# B&R Automation Studio project EFI (part 8)

### Stacker.typ
```iecst
TYPE
	StackerCtrlStatus_enum :
		(
		STACKERCTRL_STOPPED,
		STACKERCTRL_STOPPING,
		STACKERCTRL_PREPARING,
		STACKERCTRL_PREPARED,
		STACKERCTRL_PAUSING,
		STACKERCTRL_PAUSED,
		STACKERCTRL_STARTING,
		STACKERCTRL_WORKING,
		STACKERCTRL_CONTROLSTOPPING
		);
	StackerStatus_enum :
		(
		STACKER_TURNED_OFF,
		STACKER_INIT,
		STACKER_PREPARING,
		STACKER_READY,
		STACKER_WORKING,
		STACKER_FAULTED
		);
	StackerType_enum :
		(
		STACKERTY_UNDEFINED,
		STACKERTY_FULL_S,
		STACKERTY_BUNDLE_S
		);
	StackerInputs_typ : 	STRUCT
		xError : BOOL;
		xRunning : BOOL;
		xReadyToStack : BOOL;
		xFeedInterrupt : BOOL;
		xStackSuccess : BOOL;
		xRejectSuccess : BOOL;
		xModelInput : ARRAY[0..2]OF BOOL;
		Comms : StackerCommsInputs_typ;
		xStackerPresent : BOOL;
		xNoPowered : BOOL;
	END_STRUCT;
	StackerOutputs_typ : 	STRUCT
		xRun : BOOL;
		xStackEject : BOOL;
		xEjectRejectStack : BOOL;
		xPrepareToStack : BOOL;
		xRejectSheet : BOOL;
		xCleanBelts : BOOL; (*Command to empty stacker's belts*)
	END_STRUCT;
	StackerAlarms_typ : 	STRUCT
		xError : BOOL;
		xFeedInterrupt : BOOL;
		xAlrOutAutomatic : BOOL;
		xAnyAlarm : BOOL;
		xNotRemote : BOOL;
		xCriticalAlarm : BOOL;
		xWarningAlarm : BOOL;
		xNoStackerPresent : BOOL;
		xCommsError : BOOL;
		xNoPowered : BOOL;
		xBeltsStopped : BOOL;
		xRejectNoAvailable : BOOL;
		xStopRequest : BOOL; (*Stop request from Dryer when physical stop button is pressed*)
	END_STRUCT;
	StackerParametersSw_typ : 	STRUCT
		xEnabled : BOOL;
		iStackHeight : UINT;
		iStackBoardsNum : UINT;
		xStackMode : BOOL; (*(0 - Stack per number of boards, 1 - Stack per height)*)
	END_STRUCT;
	StackerParametersHw_typ : 	STRUCT
		xRejectEjectionAvailable : BOOL; (*stacker has the possibility to eject rejected boards automatically*)
		xThereIsReject : BOOL; (*Stacker has reject device*)
		rMaxSpeed : REAL := 100.0; (*Maximum speed allowed in m/min*)
		iMaxMediaWidth : UINT; (*Maximum media width allowed in mm*)
		iMinMediaWidth : UINT; (*Minimum media width allowed in mm*)
		iMinMediaThickness : UINT; (*Maximum media length allowed in mm*)
		iMaxMediaThickness : UINT; (*Minimum media length allowed in mm*)
		iMaxMediaLength : UINT; (*Maximum media length allowed in mm*)
		iMinMediaLength : UINT; (*Minimum media length allowed in mm*)
		iRejectAdjustmentDistance : INT; (*Distance in cm from beginning of the Stacker to Reject Position. Positive inside Stacker. Negative previous to Stacker*)
		iDistanceToReject : INT; (*Distance measured from "iRejectAdjusmentDistance" to reject belt start of the stacker. Physically from sensor at stacker's entry to the reject belt*)
		iMinStackHeight : UINT;
		iMaxStackHeight : UINT;
		iMinStackBoards : UINT;
		iMaxStackBoards : UINT;
		rStackerLength : REAL;
		xDoubleLineAllowed : BOOL; (*Active when allows double line printing*)
	END_STRUCT;
	StackerParameters_typ : 	STRUCT
		xInstalled : BOOL;
		xSimulationMode : BOOL; (*Defined by the configuration in Automation Studio*)
		xCommsOK : BOOL;
		xAlrPresent : BOOL;
		LineState : LineStatus_enum;
		xLineInAuto : BOOL;
		xInRemote : BOOL;
		Media : StackerMediaParameters;
		rSpeedSetPoint : REAL;
		rMediaLength : REAL;
		xPreviousDeviceStopped : BOOL;
		xDoubleLine : BOOL;
		LineStatusSummary : LineControlStatusSummarized;
		Hw : StackerParametersHw_typ;
		xActiveSlaveDiagnosis : BOOL;
	END_STRUCT;
	StackerCommands_typ : 	STRUCT
		xStart : BOOL; (*Edge commands. Reseted when managed*)
		xPrepare : BOOL; (*Edge commands. Reseted when managed*)
		xPause : BOOL; (*Edge commands. Reseted when managed*)
		xControlStop : BOOL; (*Edge commands. Reseted when managed*)
		xStop : BOOL; (*Edge commands. Reseted when managed*)
		xStartTransport : BOOL; (*Edge commands. Reseted when managed*)
		xResetAlarms : BOOL; (*Edge commands. Reseted when managed*)
		xRejectSheet : BOOL;
		xEjectPileStack : BOOL; (*Edge commands. Reseted when managed*)
		xCleanBelts : BOOL; (*Edge commands. Reseted when managed*)
		xEjectRejectStack : BOOL; (*Edge commands. Reseted when managed*)
	END_STRUCT;
	StackerOrders_typ : 	STRUCT
		xHoldReject : BOOL; (*While the signal is 1, the reject remains activated.*)
		xRejectSheet : BOOL;
		xDisableWriteBlock : BOOL; (*No read/write of channels of block (Modbus)*)
		xDisableReadBlock : BOOL;
	END_STRUCT;
	StackerDeviceStatus_typ : 	STRUCT
		xTurnedOff : BOOL;
		xInit : BOOL;
		xPreparing : BOOL;
		xReadyToStack : BOOL;
		xStacking : BOOL;
		xStackEjecting : BOOL;
		xFaulted : BOOL;
		xNotRemote : BOOL;
	END_STRUCT;
	StackerStatus_typ : 	STRUCT
		iModel : UINT; (*Model of the Device*)
		Version : EFI_version_typ;
		CtrlStatus : StackerCtrlStatus_enum;
		DeviceStatus : StackerStatus_enum;
		Device : StackerDeviceStatus_typ;
		xBeltEmpty : BOOL;
		StackerType : StackerType_enum;
		Comms : StackerCommsStatus_typ;
	END_STRUCT;
	Stacker_typ : 	STRUCT
		Inputs : StackerInputs_typ;
		Outputs : StackerOutputs_typ;
		Alarms : StackerAlarms_typ;
		ParSw : StackerParametersSw_typ;
		Parameters : StackerParameters_typ;
		Commands : StackerCommands_typ; (*Just Edge commands*)
		Orders : StackerOrders_typ;
		Status : StackerStatus_typ;
		Comms : StackerCommsOutputs_typ;
	END_STRUCT;
	StackerCommsInputs_typ : 	STRUCT
		xCommsOK : BOOL; (*Modbus communications are working properly*)
		xRemote : BOOL; (*(0: local; 1: remote)*)
		xErrorActive : BOOL; (*Any critical alarm activated*)
		xWarningActive : BOOL; (*Any warning alarm activated*)
		xOnline : BOOL; (*Modbus communications OK in stacker's side*)
		xNewFormat : BOOL; (*New box format. Please, empty stack*)
		xSerie : BOOL; (*Machine serie, SerA = 1 / SerB =0*)
		xBeltsEmpty : BOOL; (*Belts with no boards*)
		xRejectAvailable : BOOL; (*(1 = Reject Available; 0 = Reject not available)*)
		xEmergencyStopNotAcknowledged : BOOL; (*Safety alarm not acknowledge on stacker's HMI*)
		xInWorkingPosition : BOOL; (*Stacker positioned*)
		xStackExit : BOOL; (*Pile leaving*)
		xStopDemand : BOOL; (*Boards sending request*)
		xStackerEmpty : BOOL; (*Stacker and belt with no boards*)
		xStackReady : BOOL; (*Pile ready to be extracted*)
		iVersion1 : INT; (*Machine platform (Nozomi = 1)*)
		iVersion2 : INT; (*Machine project (C18000 = 0 / C14000 = 1)*)
		iVersion3 : INT; (*Hardware version*)
		iVersion4 : INT; (*Sotfware version*)
		iStatus : INT; (*Status word*)
		iAlarmWord1 : INT; (*Status word*)
		iAlarmWord2 : INT; (*Status word*)
		iAlarmWord3 : INT; (*Status word*)
		iAlarmWord4 : INT; (*Status word*)
		iAlarmWord5 : INT; (*Status word*)
		iAlarmWord6 : INT; (*Status word*)
		iAlarmWord7 : INT; (*Status word*)
		iAlarmWord8 : INT; (*Status word*)
		iAlarmWord9 : INT; (*Status word*)
		iAlarmWord10 : INT; (*Status word*)
		uiTransportSpeed : UINT;
		uiNumBoardsInCurrentPile : INT;
		uiCurrentPileHeigh : INT;
	END_STRUCT;
	StackerCommsOutputs_typ : 	STRUCT
		iControl : INT; (*Status word*)
		xBelEmpty : BOOL; (*Edge commands. Reseted when managed*)
		xResetAlarms : BOOL;
		xNewBoardParameters : BOOL; (*Pulse to let know board paramters have changed*)
		xCleanBelts : BOOL; (*Command to empty stacker's belts*)
		xEndCycle : BOOL; (*Controlled stop with pile stacked output*)
		xLastBox : BOOL; (*Signal for indicate the last box of the current pile*)
	END_STRUCT;
	StackerMediaParameters : 	STRUCT
		rThickness : REAL; (*Tile thickness to print from gui in mm*)
		rWidth : REAL; (*Board's width in mm*)
		rGap : REAL; (*Gap between boards in mm*)
		rLength : REAL; (*Board's length in mm*)
		rOffsetRegisterL1 : REAL; (*Board's width in mm*)
		rOffsetRegisterL2 : REAL; (*Board's width in mm*)
	END_STRUCT;
	StackerCommsStatus_typ : 	STRUCT
		xModuleOk : BOOL;
		ModSlaveState : UINT;
		LastError : UINT;
		LastErrorBlockNum : UINT;
		xStopButtonPressed : BOOL;
		ActOverloadError : BOOL;
		ActModbusError : BOOL;
		ActSlvConError : BOOL;
		ActRefreshError : BOOL;
		ActInternalError : BOOL;
		ActConfError : BOOL;
		HistOverloadError : BOOL;
		HistModbusError : BOOL;
		HistSlvConError : BOOL;
		HistRefreshError : BOOL;
		HistInternalError : BOOL;
		HistConfError : BOOL;
		ModbusErrorCnt : UINT;
		ModbusConErrorCnt : UINT;
		ModbusPktRefreshTimeoutCnt : UINT;
		ModbusPktPendPerSec : UINT;
		ModbusMeanResponseTime : UINT;
	END_STRUCT;
END_TYPE
```

### Program Logical/ExtPack/_Ancillaries/StackerCtrl/StackerSim/StackerSim_v1/StackerSim (IEC)

#### StackerSim.st - Init, cyclic, exit code
```iecst
PROGRAM _INIT

	Stacker ACCESS ADR(gStacker);
	SimStacker ACCESS ADR(gSimStacker);

	Stacker.Status.Comms.xModuleOk := TRUE;
	Stacker.Inputs.Comms.xBeltsEmpty:=TRUE;

END_PROGRAM

PROGRAM _CYCLIC
	(* Insert code here *)
	Stacker ACCESS ADR(gStacker);
	SimStacker ACCESS ADR(gSimStacker);

	Stacker.Inputs.xStackerPresent:=TRUE;
	Stacker.Inputs.Comms.xRemote := TRUE;

	Stacker.Inputs.xError:=SimStacker.Commands.CreateError;

	tonReady.IN:= Stacker.Outputs.xPrepareToStack;
	tonReady.PT:= T#2s;
	tonReady();
	Stacker.Inputs.xReadyToStack:=tonReady.Q;

	tonRun.IN:= Stacker.Inputs.xReadyToStack AND Stacker.Outputs.xRun;
	tonRun.PT:= T#1s;
	tonRun();
	Stacker.Inputs.xRunning:=tonRun.Q AND NOT SimStacker.Commands.StopBelts;

END_PROGRAM
```

### Library Logical/ExtPack/_Comms/ModbusComms/ModbusComms_v1/Libraries/BRSE_MB (ANSIC)

#### BRSE_MB.var
```iecst
VAR CONSTANT
	BRSE_MB_MAX_COILS : UINT := 2000;
	BRSE_MB_MAX_DISCRETE_INPUTS : UINT := 2000;
	BRSE_MB_MAX_HOLDING_REG_READ : USINT := 125;
	BRSE_MB_MAX_INPUT_REG_READ : USINT := 125;
	BRSE_MB_MAX_HOLDING_REG_WRITE : USINT := 100;
	BRSE_MB_MAX_COILS_WRITE : UINT := 800;
	BRSE_MB_ERR_REFERENCE : UINT := 20002;
	BRSE_MB_ERR_UNIT_ALLOCATED : UINT := 20001;
	BRSE_MB_ERR_ILLEGAL_FUNCTION : UINT := 1;
	BRSE_MB_ERR_ILLEGAL_DATA_ADDRESS : USINT := 2;
	BRSE_MB_ERR_ILLEGAL_DATA_VALUE : USINT := 3;
	BRSE_MB_ERR_ILLEGAL_RESPONSE_LEN : UINT := 4;
	BRSE_MB_READ_COILS : UINT := 16#01;
	BRSE_MB_READ_DISCRETE_INPUTS : UINT := 16#02;
	BRSE_MB_READ_HOLDING_REGISTERS : UINT := 16#03;
	BRSE_MB_READ_HOLDING_REG_4BYTE : UINT := 16#30;
	BRSE_MB_READ_INPUT_REGISTERS : UINT := 16#04;
	BRSE_MB_WRITE_SINGLE_COIL : UINT := 16#05;
	BRSE_MB_WRITE_SINGLE_REGISTER : UINT := 16#06;
	BRSE_MB_WRITE_MULTIPLE_COILS : UINT := 16#0F;
	BRSE_MB_WRITE_MULTIPLE_REGISTERS : UINT := 16#10;
	BRSE_MB_WRITE_MULTIPLE_REG_4BYTE : UINT := 16#31;
	BRSE_MB_ON : UINT := 16#FF00;
	BRSE_MB_OFF : UINT := 16#0000;
	BRSE_MB_MAX_UNIT_ID : USINT := 255;
	BRSE_MB_INTEL : USINT := 0; (* The server/client uses the Intel format *)
	BRSE_MB_MOTOROLA : USINT := 1; (* The server/client uses the Motorola format *)
	MB_QUEUE_SIZE : UINT := 50; (*Design parameter. Number of commands that can be queued for each client. If >= number of FB (using ClientID), race conditions (starvation?) is prevented*)
	MB_MAX_CLIENTS : USINT := 10; (*Design parameter. Maximum ClientID that can be used.*)
	MB_ERR_CLIENT_ALLOCATED : UINT := 20003; (*Error code: Queue for this client id has already been allocated*)
	MB_ERR_CLIENT_NOT_ALLOCATED : UINT := 20004; (*A request was requested from a client which hasn't been allocated*)
	MB_ERR_BUFFER : UINT := 20005; (*Buffer is too small for request or buffer address is 0*)
	MB_ERR_QUEUE_FULL : UINT := 20006;
	MB_ERR_INTERNAL : UINT := 20007;
	MB_ERR_PROTOCOL : UINT := 20008;
	MB_ERR_QUANTITY : UINT := 20009; (*Input quantity error (too big or 0)*)
	MB_ERR_CLIENT : UINT := 20010; (*Request dropped out of queue. Warm restart with remanent FUB? (Client queue is volatile)*)
	MB_ERR_CONNECTION : UINT := 20011; (*Request could not be executed: connection error or no response from server*)
END_VAR
```

#### BRSE_MB.fun
```iecst
FUNCTION MB_GetClient : UDINT (*Debug function. Returns pointer to MB_Client_typ*)
	VAR_INPUT
		ClientID : USINT;
	END_VAR
END_FUNCTION

FUNCTION BRSE_MB_Alloc : UDINT (*Allocate memory for internal data (configuration etc.). Returns error code or pointer.*)
	VAR_INPUT
		Unit : USINT; (*Unit (card id) to allocate. 0-254*)
		MaxCoils : UINT; (*Max 2000*)
		MaxHoldingRegisters : UINT; (*Max 2000*)
		MaxDiscreteInputs : UINT; (*Max 125*)
		MaxInputRegisters : UINT; (*Max 125*)
	END_VAR
END_FUNCTION

FUNCTION BRSE_MB_Coil : UINT
	VAR_INPUT
		Unit : USINT;
		Reference : UINT; (*Variable index (0-2000)*)
		VariableAddress : UDINT;
	END_VAR
END_FUNCTION

FUNCTION BRSE_MB_HoldingRegister : UINT
	VAR_INPUT
		Unit : USINT;
		Reference : UINT; (*Variable index (0-2000)*)
		VariableAddress : UDINT;
	END_VAR
END_FUNCTION

FUNCTION BRSE_MB_4ByteHoldingRegister : UINT
	VAR_INPUT
		Unit : USINT;
		Reference : UINT; (*Variable index (0-2000)*)
		VariableAddress : UDINT;
	END_VAR
END_FUNCTION

FUNCTION BRSE_MB_InputRegister : UINT
	VAR_INPUT
		Unit : USINT;
		Reference : UINT; (*Variable index (0-2000)*)
		VariableAddress : UDINT;
	END_VAR
END_FUNCTION

FUNCTION BRSE_MB_DiscreteInput : UINT
	VAR_INPUT
		Unit : USINT;
		Reference : UINT; (*Variable index (0-2000)*)
		VariableAddress : UDINT;
	END_VAR
END_FUNCTION

FUNCTION_BLOCK BRSE_MB_Server
	VAR_INPUT
		Unit : USINT;
		ClientFormat : USINT;
		InputBuffer : ARRAY[0..254] OF USINT;
	END_VAR
	VAR_OUTPUT
		OutputBuffer : ARRAY[0..254] OF USINT;
		Status : UINT;
		BufferLength : USINT; (*Total number of bytes in output buffer*)
	END_VAR
	VAR
		Request : BRSE_MB_Request_typ;
	END_VAR
END_FUNCTION_BLOCK

FUNCTION MB_AllocClient : UDINT
	VAR_INPUT
		ClientID : USINT;
	END_VAR
END_FUNCTION

FUNCTION_BLOCK MB_PollCoils
	VAR_INPUT
		ClientID : USINT;
		Enable : BOOL;
		Quantity : UINT;
		PollInterval : UDINT; (*Interval in ms between the read requests*)
		VariablesAddress : UDINT;
		StartAddress : UINT;
		Unit : USINT; (*Unit in the server*)
	END_VAR
	VAR_OUTPUT
		UpdateDone : BOOL;
		Busy : BOOL;
		Active : BOOL;
		Error : BOOL;
		ErrorID : UINT;
		Status : UINT;
	END_VAR
	VAR
		Step : UINT;
		RequestStatus : UINT;
		InternalStatus : UINT;
		RTInfo_0 : RTInfo;
		CycleTimeMs : UDINT; (*Task cycle time in ms*)
		ElapsedTime : UDINT; (*Ms since last request*)
	END_VAR
END_FUNCTION_BLOCK

FUNCTION_BLOCK MB_PollDiscreteInputs
	VAR_INPUT
		ClientID : USINT;
		Enable : BOOL;
		Quantity : UINT;
		PollInterval : UDINT; (*Interval in ms between the read requests*)
		VariablesAddress : UDINT;
		StartAddress : UINT;
		Unit : USINT; (*Unit in the server*)
	END_VAR
	VAR_OUTPUT
		UpdateDone : BOOL;
		Busy : BOOL;
		Active : BOOL;
		Error : BOOL;
		ErrorID : UINT;
		Status : UINT;
	END_VAR
	VAR
		Step : UINT;
		RequestStatus : UINT;
		InternalStatus : UINT;
		RTInfo_0 : RTInfo;
		CycleTimeMs : UDINT; (*Task cycle time in ms*)
		ElapsedTime : UDINT; (*Ms since last request*)
	END_VAR
END_FUNCTION_BLOCK

FUNCTION_BLOCK MB_PollHoldingRegisters
	VAR_INPUT
		ClientID : USINT;
		Enable : BOOL;
		Quantity : UINT;
		PollInterval : UDINT; (*Interval in ms between the read requests*)
		VariablesAddress : UDINT;
		StartAddress : UINT;
		Unit : USINT; (*Unit in the server*)
	END_VAR
	VAR_OUTPUT
		UpdateDone : BOOL;
		Busy : BOOL;
		Active : BOOL;
		Error : BOOL;
		ErrorID : UINT;
		Status : UINT;
	END_VAR
	VAR
		Step : UINT;
		RequestStatus : UINT;
		InternalStatus : UINT;
		RTInfo_0 : RTInfo;
		CycleTimeMs : UDINT; (*Task cycle time in ms*)
		ElapsedTime : UDINT; (*Ms since last request*)
	END_VAR
END_FUNCTION_BLOCK

FUNCTION_BLOCK MB_Poll4ByteHoldingRegisters
	VAR_INPUT
		ClientID : USINT;
		Enable : BOOL;
		Quantity : UINT;
		PollInterval : UDINT; (*Interval in ms between the read requests*)
		VariablesAddress : UDINT;
		StartAddress : UINT;
		Unit : USINT; (*Unit in the server*)
	END_VAR
	VAR_OUTPUT
		UpdateDone : BOOL;
		Busy : BOOL;
		Active : BOOL;
		Error : BOOL;
		ErrorID : UINT;
		Status : UINT;
	END_VAR
	VAR
		Step : UINT;
		RequestStatus : UINT;
		InternalStatus : UINT;
		RTInfo_0 : RTInfo;
		CycleTimeMs : UDINT; (*Task cycle time in ms*)
		ElapsedTime : UDINT; (*Ms since last request*)
	END_VAR
END_FUNCTION_BLOCK

FUNCTION_BLOCK MB_PollInputRegisters
	VAR_INPUT
		ClientID : USINT;
		Enable : BOOL;
		Quantity : UINT;
		PollInterval : UDINT; (*Interval in ms between the read requests*)
		VariablesAddress : UDINT;
		StartAddress : UINT;
		Unit : USINT; (*Unit in the server*)
	END_VAR
	VAR_OUTPUT
		UpdateDone : BOOL;
		Busy : BOOL;
		Active : BOOL;
		Error : BOOL;
		ErrorID : UINT;
		Status : UINT;
	END_VAR
	VAR
		Step : UINT;
		RequestStatus : UINT;
		InternalStatus : UINT;
		RTInfo_0 : RTInfo;
		CycleTimeMs : UDINT; (*Task cycle time in ms*)
		ElapsedTime : UDINT; (*Ms since last request*)
	END_VAR
END_FUNCTION_BLOCK

FUNCTION_BLOCK MB_PushCoils
	VAR_INPUT
		ClientID : USINT;
		Enable : BOOL;
		Quantity : UINT;
		PushInterval : UDINT; (*Interval in ms between the write requests*)
		VariablesAddress : UDINT;
		StartAddress : UINT;
		Unit : USINT; (*Unit in the server*)
	END_VAR
	VAR_OUTPUT
		UpdateDone : BOOL;
		Busy : BOOL;
		Active : BOOL;
		Error : BOOL;
		ErrorID : UINT;
		Status : UINT;
	END_VAR
	VAR
		Step : UINT;
		RequestStatus : UINT;
		InternalStatus : UINT;
		RTInfo_0 : RTInfo;
		CycleTimeMs : UDINT; (*Task cycle time in ms*)
		ElapsedTime : UDINT; (*Ms since last request*)
	END_VAR
END_FUNCTION_BLOCK

FUNCTION_BLOCK MB_PushHoldingRegisters
	VAR_INPUT
		ClientID : USINT;
		Enable : BOOL;
		Quantity : UINT;
		PushInterval : UDINT; (*Interval in ms between the write requests*)
		VariablesAddress : UDINT;
		StartAddress : UINT;
		Unit : USINT; (*Unit in the server*)
	END_VAR
	VAR_OUTPUT
		UpdateDone : BOOL;
		Busy : BOOL;
		Active : BOOL;
		Error : BOOL;
		ErrorID : UINT;
		Status : UINT;
	END_VAR
	VAR
		Step : UINT;
		RequestStatus : UINT;
		InternalStatus : UINT;
		RTInfo_0 : RTInfo;
		CycleTimeMs : UDINT; (*Task cycle time in ms*)
		ElapsedTime : UDINT; (*Ms since last request*)
	END_VAR
END_FUNCTION_BLOCK

FUNCTION_BLOCK MB_Push4ByteHoldingRegisters
	VAR_INPUT
		ClientID : USINT;
		Enable : BOOL;
		Quantity : UINT;
		PushInterval : UDINT; (*Interval in ms between the write requests*)
		VariablesAddress : UDINT;
		StartAddress : UINT;
		Unit : USINT; (*Unit in the server*)
	END_VAR
	VAR_OUTPUT
		UpdateDone : BOOL;
		Busy : BOOL;
		Active : BOOL;
		Error : BOOL;
		ErrorID : UINT;
		Status : UINT;
	END_VAR
	VAR
		Step : UINT;
		RequestStatus : UINT;
		InternalStatus : UINT;
		RTInfo_0 : RTInfo;
		CycleTimeMs : UDINT; (*Task cycle time in ms*)
		ElapsedTime : UDINT; (*Ms since last request*)
	END_VAR
END_FUNCTION_BLOCK

FUNCTION_BLOCK MB_ReadCoils
	VAR_INPUT
		ClientID : USINT;
		Execute : BOOL;
		Quantity : UINT;
		VariablesAddress : UDINT;
		StartAddress : UINT;
		Unit : USINT; (*Unit in the server*)
	END_VAR
	VAR_OUTPUT
		Busy : BOOL;
		Done : BOOL;
		Error : BOOL;
		ErrorID : UINT;
		Status : UINT;
	END_VAR
	VAR
		Step : UINT;
		RequestStatus : UINT;
		InternalStatus : UINT;
	END_VAR
END_FUNCTION_BLOCK

FUNCTION_BLOCK MB_ReadDiscreteInputs
	VAR_INPUT
		ClientID : USINT;
		Execute : BOOL;
		Quantity : UINT;
		VariablesAddress : UDINT;
		StartAddress : UINT;
		Unit : USINT; (*Unit in the server*)
	END_VAR
	VAR_OUTPUT
		Busy : BOOL;
		Done : BOOL;
		Error : BOOL;
		ErrorID : UINT;
		Status : UINT;
	END_VAR
	VAR
		Step : UINT;
		RequestStatus : UINT;
		InternalStatus : UINT;
	END_VAR
END_FUNCTION_BLOCK

FUNCTION_BLOCK MB_ReadHoldingRegisters
	VAR_INPUT
		ClientID : USINT;
		Execute : BOOL;
		Quantity : UINT;
		VariablesAddress : UDINT;
		StartAddress : UINT;
		Unit : USINT; (*Unit in the server*)
	END_VAR
	VAR_OUTPUT
		Busy : BOOL;
		Done : BOOL;
		Error : BOOL;
		ErrorID : UINT;
		Status : UINT;
	END_VAR
	VAR
		Step : UINT;
		RequestStatus : UINT;
		InternalStatus : UINT;
	END_VAR
END_FUNCTION_BLOCK

FUNCTION_BLOCK MB_Read4ByteHoldingRegisters
	VAR_INPUT
		ClientID : USINT;
		Execute : BOOL;
		Quantity : UINT;
		VariablesAddress : UDINT;
		StartAddress : UINT;
		Unit : USINT; (*Unit in the server*)
	END_VAR
	VAR_OUTPUT
		Busy : BOOL;
		Done : BOOL;
		Error : BOOL;
		ErrorID : UINT;
		Status : UINT;
	END_VAR
	VAR
		Step : UINT;
		RequestStatus : UINT;
		InternalStatus : UINT;
	END_VAR
END_FUNCTION_BLOCK

FUNCTION_BLOCK MB_ReadInputRegisters
	VAR_INPUT
		ClientID : USINT;
		Execute : BOOL;
		Quantity : UINT;
		VariablesAddress : UDINT;
		StartAddress : UINT;
		Unit : USINT; (*Unit in the server*)
	END_VAR
	VAR_OUTPUT
		Busy : BOOL;
		Done : BOOL;
		Error : BOOL;
		ErrorID : UINT;
		Status : UINT;
	END_VAR
	VAR
		Step : UINT;
		RequestStatus : UINT;
		InternalStatus : UINT;
	END_VAR
END_FUNCTION_BLOCK

FUNCTION_BLOCK MB_WriteCoils
	VAR_INPUT
		ClientID : USINT;
		Execute : BOOL;
		Quantity : UINT;
		VariablesAddress : UDINT;
		StartAddress : UINT;
		Unit : USINT; (*Unit in the server*)
	END_VAR
	VAR_OUTPUT
		Busy : BOOL;
		Done : BOOL;
		Error : BOOL;
		ErrorID : UINT;
		Status : UINT;
	END_VAR
	VAR
		Step : UINT;
		RequestStatus : UINT;
		InternalStatus : UINT;
	END_VAR
END_FUNCTION_BLOCK

FUNCTION_BLOCK MB_WriteHoldingRegisters
	VAR_INPUT
		ClientID : USINT;
		Execute : BOOL;
		Quantity : UINT;
		VariablesAddress : UDINT;
		StartAddress : UINT;
		Unit : USINT; (*Unit in the server*)
	END_VAR
	VAR_OUTPUT
		Busy : BOOL;
		Done : BOOL;
		Error : BOOL;
		ErrorID : UINT;
		Status : UINT;
	END_VAR
	VAR
		Step : UINT;
		RequestStatus : UINT;
		InternalStatus : UINT;
	END_VAR
END_FUNCTION_BLOCK

FUNCTION_BLOCK MB_Write4ByteHoldingRegisters
	VAR_INPUT
		ClientID : USINT;
		Execute : BOOL;
		Quantity : UINT;
		VariablesAddress : UDINT;
		StartAddress : UINT;
		Unit : USINT; (*Unit in the server*)
	END_VAR
	VAR_OUTPUT
		Busy : BOOL;
		Done : BOOL;
		Error : BOOL;
		ErrorID : UINT;
		Status : UINT;
	END_VAR
	VAR
		Step : UINT;
		RequestStatus : UINT;
		InternalStatus : UINT;
	END_VAR
END_FUNCTION_BLOCK

FUNCTION_BLOCK MB_CreateClientRequest (*This function block is used only internally and from the BRSE_MBT library (os other libraries processing the request queue)*)
	VAR_INPUT
		ClientID : USINT;
		ServerFormat : USINT;
		AdrByteBuffer : UDINT; (*Address to byte buffer where to create the request*)
		ByteBufferLen : UINT; (*Length of the byte buffer*)
	END_VAR
	VAR_OUTPUT
		RequestBufferLen : UINT; (*Length of the created modbus request. 0 means that no requests are in queue.*)
		Status : UINT; (*Error code. 0 if successful.*)
		Unit : USINT; (*Unit in the server*)
	END_VAR
END_FUNCTION_BLOCK

FUNCTION_BLOCK MB_PutClientResponse (*This function block is used only internally and from the BRSE_MBT library (os other libraries processing the request queue)*)
	VAR_INPUT
		ClientID : USINT;
		ServerFormat : USINT;
		AdrByteBuffer : UDINT;
		ByteBufferLen : UINT;
	END_VAR
	VAR_OUTPUT
		Status : UINT;
	END_VAR
	VAR
		ResponseInfo : BRSE_MB_Request_typ;
		Step : UINT;
	END_VAR
END_FUNCTION_BLOCK

FUNCTION MB_AckClientRequest : UINT (*This function is used only internally and from the BRSE_MBT library (os other libraries processing the request queue)*)
	VAR_INPUT
		ClientID : USINT;
		ReturnStatus : UINT;
	END_VAR
END_FUNCTION
```

#### Example.c
```c
/*!
\page Example

\section Example
For an example on how to use this library. Please take a look in the help for BRSE_MBT or BRSE_MBR.

*/
```

#### MB_Client.c
```c
/*! \file MB_Client.c */

#include <bur/plctypes.h>
#include "BRSE_MB.h"
#include "BRSE_MB_Main.h"

/***************************/
/* Necessary byte swapping */
/***************************/
#ifdef _SG4
	#define SWAPUINT	swapUINT
	#define SWAPINT		swapINT
#else
	#define SWAPUINT
	#define SWAPINT
#endif

#define	BUSY				65535

MB_ClientStruct_typ gMB_ClientInternal;

UDINT MB_GetClient(USINT ClientID)
{
	return gMB_ClientInternal.pClients[ClientID];
}

/*! \interface MB_AllocClient
	\brief Client: Allocate memory for internal data (request queue etc.)
	\param ClientID Client ID to allocate.
	\retval DataAddress DataAddress to internal structure. Used for debug purposes. Same value as MB_GetClient returns.
*/
UDINT MB_AllocClient(unsigned char ClientID)
{
	UINT status = 0;
	if (gMB_ClientInternal.pClients[ClientID] != 0)
	{
		return gMB_ClientInternal.pClients[ClientID];
	}
	status = TMP_alloc(sizeof(MB_Client_typ) , (void **)&(gMB_ClientInternal.pClients[ClientID]));
	if (status == 0)
	{
		memset((void *)gMB_ClientInternal.pClients[ClientID], 0, sizeof(MB_Client_typ));
	}
	else
	{
		ERRxwarning(status,(UDINT)gMB_ClientInternal.pClients[ClientID],(void *)"MBClient: No memory!");
		gMB_ClientInternal.pClients[ClientID] = 0;
	}
	return gMB_ClientInternal.pClients[ClientID];
}

void MB_CreateClientRequest(struct MB_CreateClientRequest* inst)
{
	MB_Client_typ *pQueue;
	MB_ClientQueueItem_typ *pQueueItem;
	USINT *pByteBuffer = (USINT *)inst->AdrByteBuffer;
	UINT uintSwapped;

	if (gMB_ClientInternal.pClients[inst->ClientID] == 0)
	{
		inst->Status = MB_ERR_CLIENT_NOT_ALLOCATED;
		inst->RequestBufferLen = 0;
		return;
	}
	pQueue = (MB_Client_typ *)gMB_ClientInternal.pClients[inst->ClientID];
	pQueueItem = &((*pQueue).Queue[(*pQueue).IndexExec]);
	if ((*pQueue).IndexExec == (*pQueue).IndexInsert && ((*pQueueItem).VariableAddr == 0)) /* No request in queue */
	{
		inst->Status = 0;
		inst->RequestBufferLen = 0;
		return;
	}
	else if (inst->ByteBufferLen < 5 || inst->AdrByteBuffer == 0)
	{
		inst->Status = MB_ERR_BUFFER;
		inst->RequestBufferLen = 0;
		return;
	}
	pByteBuffer[0] = (*pQueueItem).Request.Type; 					/* function code */
	uintSwapped = SWAPUINT((*pQueueItem).Request.StartAddr);
	memcpy(&(pByteBuffer[1]), &uintSwapped, 2);						/* reference number = start address */

	if(
		(*pQueueItem).Request.Type == BRSE_MB_READ_HOLDING_REG_4BYTE )
			/* 4 byte register */
	{
		pByteBuffer[0] = BRSE_MB_READ_HOLDING_REGISTERS; 					/* function code */
		uintSwapped = SWAPUINT(((*pQueueItem).Request.Quantity*2)); 		/* quantity*2 */
		memcpy(&(pByteBuffer[3]), &uintSwapped, 2);
		inst->RequestBufferLen = 5;
	}
	else if(
		(*pQueueItem).Request.Type == BRSE_MB_READ_HOLDING_REGISTERS ||
		(*pQueueItem).Request.Type == BRSE_MB_READ_COILS ||
		(*pQueueItem).Request.Type == BRSE_MB_READ_DISCRETE_INPUTS ||
		(*pQueueItem).Request.Type == BRSE_MB_READ_INPUT_REGISTERS
	)
	{
		uintSwapped = SWAPUINT((*pQueueItem).Request.Quantity); 				/* quantity */
		memcpy(&(pByteBuffer[3]), &uintSwapped, 2);
		inst->RequestBufferLen = 5;
	}
	else if ((*pQueueItem).Request.Type == BRSE_MB_WRITE_MULTIPLE_REG_4BYTE)
	{
		pByteBuffer[0] = BRSE_MB_WRITE_MULTIPLE_REGISTERS;
		uintSwapped = SWAPUINT((*pQueueItem).Request.Quantity*2); 				/* quantity *2 */
		memcpy(&(pByteBuffer[3]), &uintSwapped, 2);
		pByteBuffer[5] = (USINT) ((*pQueueItem).Request.Quantity * 4);			/* byte count *4 */
		MB_FillRegisterValues4Byte(inst->ServerFormat, pByteBuffer, pQueueItem);
		inst->RequestBufferLen = 6+4*((*pQueueItem).Request.Quantity);
	}
	else if ((*pQueueItem).Request.Type == BRSE_MB_WRITE_MULTIPLE_REGISTERS)
	{
		uintSwapped = SWAPUINT((*pQueueItem).Request.Quantity); 				/* quantity */
		memcpy(&(pByteBuffer[3]), &uintSwapped, 2);
		pByteBuffer[5] = (USINT) ((*pQueueItem).Request.Quantity * 2);			/* byte count */
		MB_FillRegisterValues(pByteBuffer, pQueueItem);
		inst->RequestBufferLen = 6+2*((*pQueueItem).Request.Quantity);
	}
	else if ((*pQueueItem).Request.Type == BRSE_MB_WRITE_SINGLE_COIL)
	{
		if(*((BOOL *)((*pQueueItem).VariableAddr)))
			pByteBuffer[3] = 0xFF;
		else
			pByteBuffer[3] = 0x00;
		pByteBuffer[4] = 0x00;
		inst->RequestBufferLen = 5;
	}
	else if ((*pQueueItem).Request.Type == BRSE_MB_WRITE_SINGLE_REGISTER)
	{
		uintSwapped = SWAPUINT(*( (INT *)((*pQueueItem).VariableAddr) ));
		memcpy(&(pByteBuffer[3]), &uintSwapped, 2);
		inst->RequestBufferLen = 5;
	}
	else if ((*pQueueItem).Request.Type == BRSE_MB_WRITE_MULTIPLE_COILS)
	{
		uintSwapped = SWAPUINT((*pQueueItem).Request.Quantity); 				/* quantity */
		memcpy(&(pByteBuffer[3]), &uintSwapped, 2);
		if (((*pQueueItem).Request.Quantity % 8) > 0)
			pByteBuffer[5] = ((*pQueueItem).Request.Quantity / 8) + 1;
		else
			pByteBuffer[5] = ((*pQueueItem).Request.Quantity / 8);
		MB_FillCoilValues(pByteBuffer, pQueueItem);
		inst->RequestBufferLen =  6+pByteBuffer[5];
	}
	inst->Unit = (*pQueueItem).Request.Unit;
}

void MB_FillRegisterValues(USINT *pByteBuffer, MB_ClientQueueItem_typ *pQueueItem)
{
	INT *pRegisterArray = (INT *)((*pQueueItem).VariableAddr);
	UINT i;
	INT intSwapped;;

	for(i=0; i<(*pQueueItem).Request.Quantity; i++)
	{
		intSwapped = SWAPINT(pRegisterArray[i]);
		memcpy(&(pByteBuffer[6 + i*2]), &intSwapped, 2);
	}
}

void MB_FillRegisterValues4Byte(USINT ServerFormat, USINT *pByteBuffer, MB_ClientQueueItem_typ *pQueueItem)
{
	INT *pRegisterArray = (INT *)((*pQueueItem).VariableAddr);
	UINT i;
	INT intSwapped;;
	if(ServerFormat == BRSE_MB_INTEL)
	{
		#ifdef _SG4
		for(i=0; i<(*pQueueItem).Request.Quantity; i++)
		{
			intSwapped = SWAPINT(pRegisterArray[i]);
			memcpy(&(pByteBuffer[6 + i*4]), &intSwapped, 2);
			intSwapped = SWAPINT(pRegisterArray[i+1]);
			memcpy(&(pByteBuffer[8 + i*4]), &intSwapped, 2);
		}
		#else
		for(i=0; i<(*pQueueItem).Request.Quantity; i++)
		{
			intSwapped = SWAPINT(pRegisterArray[i+1]);
			memcpy(&(pByteBuffer[6 + i*4]), &intSwapped, 2);
			intSwapped = SWAPINT(pRegisterArray[i]);
			memcpy(&(pByteBuffer[8 + i*4]), &intSwapped, 2);
		}
		#endif
	}
	else
	{
		#ifdef _SG4
		for(i=0; i<(*pQueueItem).Request.Quantity; i++)
		{
			intSwapped = SWAPINT(pRegisterArray[i+1]);
			memcpy(&(pByteBuffer[6 + i*4]), &intSwapped, 2);
			intSwapped = SWAPINT(pRegisterArray[i]);
			memcpy(&(pByteBuffer[8 + i*4]), &intSwapped, 2);
		}
		#else
		for(i=0; i<(*pQueueItem).Request.Quantity; i++)
		{
			intSwapped = SWAPINT(pRegisterArray[i]);
			memcpy(&(pByteBuffer[6 + i*4]), &intSwapped, 2);
			intSwapped = SWAPINT(pRegisterArray[i+1]);
			memcpy(&(pByteBuffer[8 + i*4]), &intSwapped, 2);
		}
		#endif
	}
}

void MB_PutRegisterValues(USINT *pByteBuffer, MB_ClientQueueItem_typ *pQueueItem)
{
	INT *pRegisterArray = (INT *)((*pQueueItem).VariableAddr);
	UINT i;
	INT intSwapped;

	for(i=0; i<(*pQueueItem).Request.Quantity; i++)
	{
		memcpy(&(intSwapped), &(pByteBuffer[2 + i*2]), 2);
		pRegisterArray[i] = SWAPINT(intSwapped);
	}

}

void MB_PutRegisterValues4Byte(USINT ServerFormat,USINT *pByteBuffer, MB_ClientQueueItem_typ *pQueueItem)
{
	INT *pRegisterArray = (INT *)((*pQueueItem).VariableAddr);
	UINT i;
	INT intSwapped;

	if(ServerFormat == BRSE_MB_INTEL)
	{
		#ifdef _SG4
		for(i=0; i<(*pQueueItem).Request.Quantity; i++)
		{
			memcpy(&(intSwapped), &(pByteBuffer[2 + i*4]), 2);
			pRegisterArray[i*2] = SWAPINT(intSwapped);
			memcpy(&(intSwapped), &(pByteBuffer[4 + i*4]), 2);
			pRegisterArray[i*2+1] = SWAPINT(intSwapped);
		}
		#else
		for(i=0; i<(*pQueueItem).Request.Quantity; i++)
		{
			memcpy(&(intSwapped), &(pByteBuffer[2 + i*4]), 2);
			pRegisterArray[i*2+1] = SWAPINT(intSwapped);
			memcpy(&(intSwapped), &(pByteBuffer[4 + i*4]), 2);
			pRegisterArray[i*2] = SWAPINT(intSwapped);
		}
		#endif
	}
	else
	{
		#ifdef _SG4
		for(i=0; i<(*pQueueItem).Request.Quantity; i++)
		{
			memcpy(&(intSwapped), &(pByteBuffer[2 + i*4]), 2);
			pRegisterArray[i*2+1] = SWAPINT(intSwapped);
			memcpy(&(intSwapped), &(pByteBuffer[4 + i*4]), 2);
			pRegisterArray[i*2] = SWAPINT(intSwapped);
		}
		#else
		for(i=0; i<(*pQueueItem).Request.Quantity; i++)
		{
			memcpy(&(intSwapped), &(pByteBuffer[2 + i*4]), 2);
			pRegisterArray[i*2] = SWAPINT(intSwapped);
			memcpy(&(intSwapped), &(pByteBuffer[4 + i*4]), 2);
			pRegisterArray[i*2+1] = SWAPINT(intSwapped);
		}
		#endif
	}

}

void MB_FillCoilValues(USINT *pByteBuffer, MB_ClientQueueItem_typ *pQueueItem)
{
	BOOL *pCoilArray = (BOOL *)((*pQueueItem).VariableAddr);
	UINT i;

	for(i=0; i<(*pQueueItem).Request.Quantity; i++)
	{
		if(pCoilArray[i])
			pByteBuffer[6 + (i/8)] = pByteBuffer[6 + (i/8)] | (USINT)(0x01 << (i%8));
		else
			pByteBuffer[6 + (i/8)] = pByteBuffer[6 + (i/8)] & (USINT)~(0x01 << (i%8));
	}
}

void MB_PutCoilValues(USINT *pByteBuffer, MB_ClientQueueItem_typ *pQueueItem)
{
	BOOL *pCoilArray = (BOOL *)((*pQueueItem).VariableAddr);
	UINT i;

	for(i=0; i < (*pQueueItem).Request.Quantity; i++)
	{
		if ((pByteBuffer[2 + (i/8)] & (USINT)(0x01 << (i%8))))
			pCoilArray[i] = 1;
		else
			pCoilArray[i] = 0;
	}
}

/**/
void MB_PutClientResponse(struct MB_PutClientResponse* inst)
{
	USINT *pByteBuffer = (USINT *)inst->AdrByteBuffer;
	UINT uintSwapped;
	UINT returnStatus;
	MB_Client_typ *pQueue;
	MB_ClientQueueItem_typ *pQueueItem;

	/*****************************/
	/* Parse response information */
	/*****************************/
	if (gMB_ClientInternal.pClients[inst->ClientID] == 0)
	{
		inst->Status = MB_ERR_CLIENT_NOT_ALLOCATED;
		return;
	}

	pQueue = (MB_Client_typ *)gMB_ClientInternal.pClients[inst->ClientID];
	pQueueItem = &((*pQueue).Queue[(*pQueue).IndexExec]);

	inst->Status = BUSY;

	inst->ResponseInfo.Type = pByteBuffer[0]; 	/* Function code (byte 0) */

	/*special case using 4 byte holding registers*/
	if
	(
		(
			(inst->ResponseInfo.Type == BRSE_MB_READ_HOLDING_REGISTERS)
			&&
			((*pQueueItem).Request.Type == BRSE_MB_READ_HOLDING_REG_4BYTE)
		)
		||
		(
			(inst->ResponseInfo.Type == BRSE_MB_WRITE_MULTIPLE_REGISTERS)
			&&
			((*pQueueItem).Request.Type == BRSE_MB_WRITE_MULTIPLE_REG_4BYTE)
		)
	)
	{
		inst->ResponseInfo.Type = (*pQueueItem).Request.Type;
	}

	if (inst->ResponseInfo.Type >= 0x80)		/* Modbus error */
	{
		returnStatus = pByteBuffer[1];
	}
	else if (inst->ResponseInfo.Type != (*pQueueItem).Request.Type)
	{
		returnStatus = MB_ERR_PROTOCOL;
	}
	else if (inst->ResponseInfo.Type == 0) /* FC 0 does not exist */
	{
		returnStatus = MB_ERR_PROTOCOL;
	}
	else
	{
		if (inst->ResponseInfo.Type == BRSE_MB_WRITE_MULTIPLE_REG_4BYTE ||
			inst->ResponseInfo.Type == BRSE_MB_WRITE_MULTIPLE_REGISTERS ||
			inst->ResponseInfo.Type == BRSE_MB_WRITE_MULTIPLE_COILS)
		{
			memcpy(&uintSwapped, &pByteBuffer[1], 2);				/* Reference number (byte 1,2) */
			inst->ResponseInfo.StartAddr = SWAPUINT(uintSwapped);
			memcpy(&uintSwapped, &pByteBuffer[3], 2);
			inst->ResponseInfo.Quantity = SWAPUINT(uintSwapped);	/* Quantity */
			returnStatus = 0;
		}
		else if (inst->ResponseInfo.Type == BRSE_MB_READ_HOLDING_REG_4BYTE)
		{
			inst->ResponseInfo.Quantity = pByteBuffer[1]/4; /* byte count */
			MB_PutRegisterValues4Byte(inst->ServerFormat, pByteBuffer, pQueueItem);
			returnStatus = 0;
		}
		else if (inst->ResponseInfo.Type == BRSE_MB_READ_HOLDING_REGISTERS ||
			inst->ResponseInfo.Type == BRSE_MB_READ_INPUT_REGISTERS)
		{
			inst->ResponseInfo.Quantity = pByteBuffer[1]/2; /* byte count / 2 */
			MB_PutRegisterValues(pByteBuffer, pQueueItem);
			returnStatus = 0;
		}
		else if (inst->ResponseInfo.Type == BRSE_MB_READ_COILS ||
			inst->ResponseInfo.Type == BRSE_MB_READ_DISCRETE_INPUTS)
		{
			inst->ResponseInfo.Quantity = (*pQueueItem).Request.Quantity; /* number of coils / inputs */
			MB_PutCoilValues(pByteBuffer, pQueueItem);
			returnStatus = 0;
		}
		else if (inst->ResponseInfo.Type == BRSE_MB_WRITE_SINGLE_COIL ||
			inst->ResponseInfo.Type == BRSE_MB_WRITE_SINGLE_REGISTER)
		{
			memcpy(&uintSwapped, &pByteBuffer[1], 2);				/* Reference number (byte 1,2) */
			inst->ResponseInfo.StartAddr = SWAPUINT(uintSwapped);
			returnStatus = 0;
		}
		else
		{
			returnStatus = MB_ERR_PROTOCOL;
		}
	}
	MB_AckClientRequest(inst->ClientID, returnStatus);
	inst->Status = returnStatus;
}
```

#### MB_ModbusClientFunctions.c
```c
/*! \file MB_ModbusClientFunctions.c */

#include <bur/plctypes.h>
#include "BRSE_MB.h"
#include "BRSE_MB_Main.h"

#define	BUSY				65535

extern MB_ClientStruct_typ gMB_ClientInternal;

UINT MB_AddToRequestQueue(USINT clientID, USINT fc, UINT quantity, UINT startAddress, UDINT variableAddress, UDINT statusAddress, USINT Unit);

/***
 * This macro is the code basis for all non-cyclic modbus function calls from the application.
 * The only thing that differs is the function code.
 */
#define EXEC_MODBUS_FUNCTION_MACRO(functionCode)	\
		switch(inst->Step)							\
		{											\
			case 0: /* idle */						\
				if (inst->Done || inst->Error)		\
				{	/*reset out signals */			\
					inst->Done = inst->Execute;		\
					inst->Error = inst->Execute;	\
				}									\
				else if (inst->Execute)				\
				{									\
					inst->Step = 1;					\
				}									\
				inst->Busy = 0;						\
				break;								\
													\
			case 1:	/* add req to queue */			\
				inst->InternalStatus = MB_AddToRequestQueue(inst->ClientID, functionCode, inst->Quantity, inst->StartAddress, inst->VariablesAddress, (UDINT)&(inst->RequestStatus), inst->Unit); \
				if (inst->InternalStatus == 0)		\
				{									\
					inst->Status = BUSY;			\
					inst->Step = 2;					\
				}									\
				else								\
				{									\
					inst->Status = inst->InternalStatus; \
				}									\
				inst->Error = 0;					\
				inst->Done = 0;						\
				inst->Busy = 1;						\
				break;								\
													\
			case 2:									\
				if (inst->RequestStatus == 0) 		\
				{									\
					inst->Status = 0;				\
					inst->Done = 1;					\
					inst->Error = 0;				\
					inst->Busy = 0;					\
					inst->Step = 0;					\
				}									\
				else if (inst->RequestStatus != BUSY) 	\
				{									\
					inst->Status = inst->RequestStatus; \
					inst->Done = 0;					\
					inst->Error = 1;				\
					inst->Busy = 0;					\
					inst->Step = 0;					\
				}									\
				else if (MB_QueueStatus(inst->ClientID) == 0)	\
				{									\
					inst->Status = MB_ERR_CLIENT;	\
					ERRxwarning(58001,inst->ClientID,(void *)"MB_Client_Fub: No client queue!");\
					inst->Done = 0;					\
					inst->Error = 1;				\
					inst->Busy = 0;					\
					inst->Step = 0;					\
				}									\
				break;								\
		}

/*
 * This macro is the code basis for all cyclic modbus function calls from the application.
 * The only thing that differs is the function code.
 *
 * The functions places the request in queue and waits for the request to be executed.
 * When the function has been executed, the resulting status is set in the inst->RequestStatus variable.
 * 0 if successful.
 */
#define EXEC_MODBUS_CYCLIC_FUNCTION_MACRO(functionCode, interval) 	\
		if (!inst->Enable)									\
		{													\
			inst->Active = 0;								\
			inst->Busy = 0;									\
			inst->UpdateDone = 0;							\
			inst->Status = 0;								\
			return;											\
		}													\
		inst->ElapsedTime += inst->CycleTimeMs;				\
		switch(inst->Step)									\
		{													\
			case 0: /* init cycle time */					\
				inst->Status = 0;							\
				inst->RTInfo_0.enable = 1;					\
				RTInfo(&inst->RTInfo_0);					\
				if (inst->RTInfo_0.status == 0)				\
				{											\
					inst->CycleTimeMs = inst->RTInfo_0.cycle_time/1000;\
					inst->Step = 2; /* go directly to first push/poll */\
				}											\
				break;										\
															\
			case 1: /* idle */								\
				if (inst->ElapsedTime >= interval) 			\
				{											\
					inst->Step = 2;							\
					inst->ElapsedTime = 0; /*reset*/		\
				}											\
				else										\
					break;									\
															\
			case 2:	 /* put request in queue */				\
				inst->UpdateDone = 0;						\
				inst->InternalStatus = MB_AddToRequestQueue(inst->ClientID, functionCode, inst->Quantity, inst->StartAddress, inst->VariablesAddress, (UDINT)&(inst->RequestStatus), inst->Unit); \
				if (inst->InternalStatus == 0)				\
				{											\
					inst->Step = 3;							\
					inst->Status = BUSY;					\
				}											\
				else										\
				{											\
					inst->Status = inst->InternalStatus;	\
				}											\
				break;										\
															\
			case 3: /* await request finished */			\
				inst->Status = BUSY;						\
				if (inst->RequestStatus == 0) /* finished */\
				{											\
					inst->UpdateDone = 1;					\
					inst->Status = 0;						\
					inst->Step = 1;							\
				}											\
				else if (inst->RequestStatus != BUSY) /* finished with errors */\
				{											\
					inst->Status = inst->RequestStatus;		\
					inst->Step = 1;							\
				}											\
				else if (MB_QueueStatus(inst->ClientID) == 0)\
				{											\
					inst->Status = MB_ERR_CLIENT;			\
					ERRxwarning(58002,inst->ClientID,(void *)"MB_Client_Fub: No client queue!");\
					inst->Step = 1;							\
				}											\
				break;										\
		}													\
		inst->Active = (inst->Enable && inst->Step != 0) ? 1 : 0; \
		inst->Error = (inst->Status != 0 && inst->Status != BUSY) ? 1 : 0; \
		inst->ErrorID = (inst->Status < 5) ? inst->Status : 0; /* only modbus protocol errors */\
		inst->Busy = (inst->Status == BUSY) ? 1 : 0;

#define CHECK_INPUT_QUANTITY_MACRO(maxQuantity) 										\
		if(inst->Quantity > maxQuantity || inst->Quantity == 0) 						\
		{																				\
			inst->Status = MB_ERR_QUANTITY;												\
			inst->Done = 0;																\
			inst->Error = 1;															\
			inst->ErrorID = 0; 															\
			inst->Busy = 0;																\
			return;																		\
		}

#define CHECK_INPUT_QUANTITY_CYCLIC_MACRO(maxQuantity) 									\
		if(inst->Quantity > maxQuantity || inst->Quantity == 0) 						\
		{																				\
			inst->Status = MB_ERR_QUANTITY;												\
			inst->Active = 0;															\
			inst->Error = 1;															\
			inst->ErrorID = 0; 															\
			inst->Busy = 0;																\
			inst->UpdateDone = 0;														\
			return;																		\
		}

/*
 *
 */

/*! \interface MB_WriteHoldingRegisters
	\brief Client: Write event triggered to a holding register

	\param[in] 	ClientID	Identity created in AllocClient.
	\param[in]	Execute	Enables execution.
	\param[in]	Quantity	Number of register to write to.
	\param[in]	VariablesAddress	Address of the integer variable.
	\param[in]	StartAddress	Address in the server to write to.
	\param[in] 	Unit	Identity of the unit (0-255) in the server.
	\param[out] Busy	Set to TRUE when function are busy.
	\param[out] Done	When the function has completed succesfully, this value is set to TRUE.
	\param[out] Error	If an error occurs while exeuting the function, this output is set to TRUE.
	\param[out] ErrorID	Error number from the function block.
	\param[out] Status	Normally set to zero otherwise something is wrong or function are waiting to get completed.
*/
void MB_WriteHoldingRegisters(struct MB_WriteHoldingRegisters* inst)
{
	CHECK_INPUT_QUANTITY_MACRO(BRSE_MB_MAX_HOLDING_REG_WRITE)
	EXEC_MODBUS_FUNCTION_MACRO(inst->Quantity == 1 ? BRSE_MB_WRITE_SINGLE_REGISTER : BRSE_MB_WRITE_MULTIPLE_REGISTERS)
}

/*! \interface MB_Write4ByteHoldingRegisters
	\brief Client: Write event triggered to a 4 byte register using 2 holding registers

	\param[in] 	ClientID	Identity created in AllocClient.
	\param[in]	Execute	Enables execution.
	\param[in]	Quantity	Number of 4-byte variables to write to. Corresponds to the double amount of holding registers.
	\param[in]	VariablesAddress	Address of the 4 byte variable.
	\param[in]	StartAddress	Address in the server to write to.
	\param[in] 	Unit	Identity of the unit (0-255) in the server.
	\param[out] Busy	Set to TRUE when function are busy.
	\param[out] Done	When the function has completed succesfully, this value is set to TRUE.
	\param[out] Error	If an error occurs while exeuting the function, this output is set to TRUE.
	\param[out] ErrorID	Error number from the function block.
	\param[out] Status	Normally set to zero otherwise something is wrong or function are waiting to get completed.
*/
void MB_Write4ByteHoldingRegisters(struct MB_Write4ByteHoldingRegisters* inst)
{
	CHECK_INPUT_QUANTITY_MACRO(BRSE_MB_MAX_HOLDING_REG_WRITE)
	EXEC_MODBUS_FUNCTION_MACRO(BRSE_MB_WRITE_MULTIPLE_REG_4BYTE)
}

/*! \interface MB_WriteCoils
	\brief Client: Write event triggered to a coil

	\param[in] 	ClientID	Identity created in AllocClient.
	\param[in]	Execute	Enables execution.
	\param[in]	Quantity	Number of register to write to.
	\param[in]	VariablesAddress	Address of the bool variable.
	\param[in]	StartAddress	Address in the server to write to.
	\param[in] 	Unit	Identity of the unit (0-255) in the server.
	\param[out] Busy	Set to TRUE when function are busy.
	\param[out] Done	When the function has completed succesfully, this value is set to TRUE.
	\param[out] Error	If an error occurs while exeuting the function, this output is set to TRUE.
	\param[out] ErrorID	Error number from the function block.
	\param[out] Status	Normally set to zero otherwise something is wrong or function are waiting to get completed.
*/
void MB_WriteCoils(struct MB_WriteCoils* inst)
{
	CHECK_INPUT_QUANTITY_MACRO(BRSE_MB_MAX_COILS_WRITE)
	EXEC_MODBUS_FUNCTION_MACRO(inst->Quantity == 1 ? BRSE_MB_WRITE_SINGLE_COIL : BRSE_MB_WRITE_MULTIPLE_COILS)
}

/*! \interface MB_ReadHoldingRegisters
	\brief Client: Read event triggered from a holding register

	\param[in] 	ClientID	Identity created in AllocClient.
	\param[in]	Execute	Enables execution.
	\param[in]	Quantity	Number of register to read from.
	\param[in]	VariablesAddress	Address of the integer variable.
	\param[in]	StartAddress	Address in the server to read from.
	\param[in] 	Unit	Identity of the unit (0-255) in the server.
	\param[out] Busy	Set to TRUE when function are busy.
	\param[out] Done	When the function has completed succesfully, this value is set to TRUE.
	\param[out] Error	If an error occurs while exeuting the function, this output is set to TRUE.
	\param[out] ErrorID	Error number from the function block.
	\param[out] Status	Normally set to zero otherwise something is wrong or function are waiting to get completed.
*/
void MB_ReadHoldingRegisters(struct MB_ReadHoldingRegisters* inst)
{
	CHECK_INPUT_QUANTITY_MACRO(BRSE_MB_MAX_HOLDING_REG_READ)
	EXEC_MODBUS_FUNCTION_MACRO(BRSE_MB_READ_HOLDING_REGISTERS)
}

/*! \interface MB_Read4ByteHoldingRegisters
	\brief Client: Read event triggered from a 4 byte register using 2 holding registers

	\param[in] 	ClientID	Identity created in AllocClient.
	\param[in]	Execute	Enables execution.
	\param[in]	Quantity	Number of 4-byte variables to read. Corresponds to the double amount of holding registers.
	\param[in]	VariablesAddress	Address of the 4 byte variable.
	\param[in]	StartAddress	Address in the server to read from.
	\param[in] 	Unit	Identity of the unit (0-255) in the server.
	\param[out] Busy	Set to TRUE when function are busy.
	\param[out] Done	When the function has completed succesfully, this value is set to TRUE.
	\param[out] Error	If an error occurs while exeuting the function, this output is set to TRUE.
	\param[out] ErrorID	Error number from the function block.
	\param[out] Status	Normally set to zero otherwise something is wrong or function are waiting to get completed.
*/
void MB_Read4ByteHoldingRegisters(struct MB_Read4ByteHoldingRegisters* inst)
{
	CHECK_INPUT_QUANTITY_MACRO(BRSE_MB_MAX_HOLDING_REG_READ)
	EXEC_MODBUS_FUNCTION_MACRO(BRSE_MB_READ_HOLDING_REG_4BYTE)
}

/*! \interface MB_ReadCoils
	\brief Client: Read event triggered from a coil

	\param[in] 	ClientID	Identity created in AllocClient.
	\param[in]	Execute	Enables execution.
	\param[in]	Quantity	Number of register to read from.
	\param[in]	VariablesAddress	Address of the bool variable.
	\param[in]	StartAddress	Address in the server to read from.
	\param[in] 	Unit	Identity of the unit (0-255) in the server.
	\param[out] Busy	Set to TRUE when function are busy.
	\param[out] Done	When the function has completed succesfully, this value is set to TRUE.
	\param[out] Error	If an error occurs while exeuting the function, this output is set to TRUE.
	\param[out] ErrorID	Error number from the function block.
	\param[out] Status	Normally set to zero otherwise something is wrong or function are waiting to get completed.
*/
void MB_ReadCoils(struct MB_ReadCoils* inst)
{
	CHECK_INPUT_QUANTITY_MACRO(BRSE_MB_MAX_COILS)
	EXEC_MODBUS_FUNCTION_MACRO(BRSE_MB_READ_COILS)
}

/*! \interface MB_ReadInputRegisters
	\brief Client: Read event triggered from a input register

	\param[in] 	ClientID	Identity created in AllocClient.
	\param[in]	Execute	Enables execution.
	\param[in]	Quantity	Number of register to read from.
	\param[in]	VariablesAddress	Address of the integer variable.
	\param[in]	StartAddress	Address in the server to read from.
	\param[in] 	Unit	Identity of the unit (0-255) in the server.
	\param[out] Busy	Set to TRUE when function are busy.
	\param[out] Done	When the function has completed succesfully, this value is set to TRUE.
	\param[out] Error	If an error occurs while exeuting the function, this output is set to TRUE.
	\param[out] ErrorID	Error number from the function block.
	\param[out] Status	Normally set to zero otherwise something is wrong or function are waiting to get completed.
*/
void MB_ReadInputRegisters(struct MB_ReadInputRegisters* inst)
{
	CHECK_INPUT_QUANTITY_MACRO(BRSE_MB_MAX_INPUT_REG_READ)
	EXEC_MODBUS_FUNCTION_MACRO(BRSE_MB_READ_INPUT_REGISTERS)
}

/*! \interface MB_ReadDiscreteInputs
	\brief Client: Read event triggered from a discreate input

	\param[in] 	ClientID	Identity created in AllocClient.
	\param[in]	Execute	Enables execution.
	\param[in]	Quantity	Number of register to read from.
	\param[in]	VariablesAddress	Address of the bool variable.
	\param[in]	StartAddress	Address in the server to read from.
	\param[in] 	Unit	Identity of the unit (0-255) in the server.
	\param[out] Busy	Set to TRUE when function are busy.
	\param[out] Done	When the function has completed succesfully, this value is set to TRUE.
	\param[out] Error	If an error occurs while exeuting the function, this output is set to TRUE.
	\param[out] ErrorID	Error number from the function block.
	\param[out] Status	Normally set to zero otherwise something is wrong or function are waiting to get completed.
*/
void MB_ReadDiscreteInputs(struct MB_ReadDiscreteInputs* inst)
{
	CHECK_INPUT_QUANTITY_MACRO(BRSE_MB_MAX_DISCRETE_INPUTS)
	EXEC_MODBUS_FUNCTION_MACRO(BRSE_MB_READ_DISCRETE_INPUTS)
}

/*! \interface MB_PushHoldingRegisters
	\brief Client: Write cyclic to a holding register

	\param[in] 	ClientID	Identity created in AllocClient.
	\param[in]	Enable	Enables execution.
	\param[in]	Quantity	Number of register to write to.
	\param[in]	PushInterval	Interval in ms between the Write requests.
	\param[in]	VariablesAddress	Address of the integer variable.
	\param[in]	StartAddress	Address in the server to write to.
	\param[in] 	Unit	Identity of the unit (0-255) in the server.
	\param[out] UpdateDone	When the function has completed succesfully, this value is set to TRUE.
	\param[out] Active	Set to TRUE when function is active.
	\param[out] Busy	Set to TRUE when function is accessing the server.
	\param[out] Error	If an error occurs while exeuting the function, this output is set to TRUE.
	\param[out] ErrorID	Error number from the function block.
	\param[out] Status	Normally set to zero otherwise something is wrong or function are waiting to get completed.
*/
void MB_PushHoldingRegisters(struct MB_PushHoldingRegisters* inst)
{
	CHECK_INPUT_QUANTITY_CYCLIC_MACRO(BRSE_MB_MAX_HOLDING_REG_WRITE)
	EXEC_MODBUS_CYCLIC_FUNCTION_MACRO((inst->Quantity == 1) ? BRSE_MB_WRITE_SINGLE_REGISTER : BRSE_MB_WRITE_MULTIPLE_REGISTERS, inst->PushInterval)
}

/*! \interface MB_Push4ByteHoldingRegisters
	\brief Client: Write cyclic to a 4 byte register using 2 holding registers

	\param[in] 	ClientID	Identity created in AllocClient.
	\param[in]	Enable	Enables execution.
	\param[in]	Quantity	Number of 4-byte variables to write to. Corresponds to the double amount of holding registers.
	\param[in]	PushInterval	Interval in ms between the Write requests.
	\param[in]	VariablesAddress	Address of the 4 byte variable.
	\param[in]	StartAddress	Address in the server to write to.
	\param[in] 	Unit	Identity of the unit (0-255) in the server.
	\param[out] UpdateDone	When the function has completed succesfully, this value is set to TRUE.
	\param[out] Active	Set to TRUE when function is active.
	\param[out] Busy	Set to TRUE when function is accessing the server.
	\param[out] Error	If an error occurs while exeuting the function, this output is set to TRUE.
	\param[out] ErrorID	Error number from the function block.
	\param[out] Status	Normally set to zero otherwise something is wrong or function are waiting to get completed.
*/
void MB_Push4ByteHoldingRegisters(struct MB_Push4ByteHoldingRegisters* inst)
{
	CHECK_INPUT_QUANTITY_CYCLIC_MACRO(BRSE_MB_MAX_HOLDING_REG_WRITE)
	EXEC_MODBUS_CYCLIC_FUNCTION_MACRO(BRSE_MB_WRITE_MULTIPLE_REG_4BYTE, inst->PushInterval)
}

/*! \interface MB_PushCoils
	\brief Client: Write cyclic to a coil

	\param[in] 	ClientID	Identity created in AllocClient.
	\param[in]	Enable	Enables execution.
	\param[in]	Quantity	Number of register to write to.
	\param[in]	PushInterval	Interval in ms between the Write requests.
	\param[in]	VariablesAddress	Address of the bool variable.
	\param[in]	StartAddress	Address in the server to write to.
	\param[in] 	Unit	Identity of the unit (0-255) in the server.
	\param[out] UpdateDone	When the function has completed succesfully, this value is set to TRUE.
	\param[out] Active	Set to TRUE when function is active.
	\param[out] Busy	Set to TRUE when function is accessing the server.
	\param[out] Error	If an error occurs while exeuting the function, this output is set to TRUE.
	\param[out] ErrorID	Error number from the function block.
	\param[out] Status	Normally set to zero otherwise something is wrong or function are waiting to get completed.
*/
void MB_PushCoils(struct MB_PushCoils* inst)
{
	CHECK_INPUT_QUANTITY_CYCLIC_MACRO(BRSE_MB_MAX_COILS_WRITE)
	EXEC_MODBUS_CYCLIC_FUNCTION_MACRO(inst->Quantity == 1 ? BRSE_MB_WRITE_SINGLE_COIL : BRSE_MB_WRITE_MULTIPLE_COILS, inst->PushInterval)
}

/*! \interface MB_PollHoldingRegisters
	\brief Client: Read cyclic from a holding register

	\param[in] 	ClientID	Identity created in AllocClient.
	\param[in]	Enable	Enables execution.
	\param[in]	Quantity	Number of register to read from.
	\param[in]	PollInterval	Interval in ms between the Read requests.
	\param[in]	VariablesAddress	Address of the integer variable.
	\param[in]	StartAddress	Address in the server to read from.
	\param[in] 	Unit	Identity of the unit (0-255) in the server.
	\param[out] UpdateDone	When the function has completed succesfully, this value is set to TRUE.
	\param[out] Active	Set to TRUE when function is active.
	\param[out] Busy	Set to TRUE when function is accessing the server.
	\param[out] Error	If an error occurs while exeuting the function, this output is set to TRUE.
	\param[out] ErrorID	Error number from the function block.
	\param[out] Status	Normally set to zero otherwise something is wrong or function are waiting to get completed.
*/
void MB_PollHoldingRegisters(struct MB_PollHoldingRegisters* inst)
{
	CHECK_INPUT_QUANTITY_CYCLIC_MACRO(BRSE_MB_MAX_HOLDING_REG_READ)
	EXEC_MODBUS_CYCLIC_FUNCTION_MACRO(BRSE_MB_READ_HOLDING_REGISTERS, inst->PollInterval)
}

/*! \interface MB_Poll4ByteHoldingRegisters
	\brief Client: Read cyclic from a 4 byte register using 2 holding registers

	\param[in] 	ClientID	Identity created in AllocClient.
	\param[in]	Enable	Enables execution.
	\param[in]	Quantity	Number of 4-byte variables to read. Corresponds to the double amount of holding registers.
	\param[in]	PollInterval	Interval in ms between the Read requests.
	\param[in]	VariablesAddress	Address of the 4 byte variable.
	\param[in]	StartAddress	Address in the server to read from.
	\param[in] 	Unit	Identity of the unit (0-255) in the server.
	\param[out] UpdateDone	When the function has completed succesfully, this value is set to TRUE.
	\param[out] Active	Set to TRUE when function is active.
	\param[out] Busy	Set to TRUE when function is accessing the server.
	\param[out] Error	If an error occurs while exeuting the function, this output is set to TRUE.
	\param[out] ErrorID	Error number from the function block.
	\param[out] Status	Normally set to zero otherwise something is wrong or function are waiting to get completed.
*/
void MB_Poll4ByteHoldingRegisters(struct MB_Poll4ByteHoldingRegisters* inst)
{
	CHECK_INPUT_QUANTITY_CYCLIC_MACRO(BRSE_MB_MAX_HOLDING_REG_READ)
	EXEC_MODBUS_CYCLIC_FUNCTION_MACRO(BRSE_MB_READ_HOLDING_REG_4BYTE, inst->PollInterval)
}

/*! \interface MB_PollCoils
	\brief Client: Read cyclic from a coil

	\param[in] 	ClientID	Identity created in AllocClient.
	\param[in]	Enable	Enables execution.
	\param[in]	Quantity	Number of register to read from.
	\param[in]	PollInterval	Interval in ms between the Read requests.
	\param[in]	VariablesAddress	Address of the bool variable.
	\param[in]	StartAddress	Address in the server to read from.
	\param[in] 	Unit	Identity of the unit (0-255) in the server.
	\param[out] UpdateDone	When the function has completed succesfully, this value is set to TRUE.
	\param[out] Active	Set to TRUE when function is active.
	\param[out] Busy	Set to TRUE when function is accessing the server.
	\param[out] Error	If an error occurs while exeuting the function, this output is set to TRUE.
	\param[out] ErrorID	Error number from the function block.
	\param[out] Status	Normally set to zero otherwise something is wrong or function are waiting to get completed.
*/
void MB_PollCoils(struct MB_PollCoils* inst)
{
	CHECK_INPUT_QUANTITY_CYCLIC_MACRO(BRSE_MB_MAX_COILS)
	EXEC_MODBUS_CYCLIC_FUNCTION_MACRO(BRSE_MB_READ_COILS, inst->PollInterval)
}

/*! \interface MB_PollInputRegisters
	\brief Client: Read cyclic from a input register

	\param[in] 	ClientID	Identity created in AllocClient.
	\param[in]	Enable	Enables execution.
	\param[in]	Quantity	Number of register to read from.
	\param[in]	PollInterval	Interval in ms between the Read requests.
	\param[in]	VariablesAddress	Address of the integer variable.
	\param[in]	StartAddress	Address in the server to read from.
	\param[in] 	Unit	Identity of the unit (0-255) in the server.
	\param[out] UpdateDone	When the function has completed succesfully, this value is set to TRUE.
	\param[out] Active	Set to TRUE when function is active.
	\param[out] Busy	Set to TRUE when function is accessing the server.
	\param[out] Error	If an error occurs while exeuting the function, this output is set to TRUE.
	\param[out] ErrorID	Error number from the function block.
	\param[out] Status	Normally set to zero otherwise something is wrong or function are waiting to get completed.
*/
void MB_PollInputRegisters(struct MB_PollInputRegisters* inst)
{
	CHECK_INPUT_QUANTITY_CYCLIC_MACRO(BRSE_MB_MAX_INPUT_REG_READ)
	EXEC_MODBUS_CYCLIC_FUNCTION_MACRO(BRSE_MB_READ_INPUT_REGISTERS, inst->PollInterval)
}

/*! \interface MB_PollDiscreteInputs
	\brief Client: Read cyclic from a discreate input

	\param[in] 	ClientID	Identity created in AllocClient.
	\param[in]	Enable	Enables execution.
	\param[in]	Quantity	Number of register to read from.
	\param[in]	PollInterval	Interval in ms between the Read requests.
	\param[in]	VariablesAddress	Address of the bool variable.
	\param[in]	StartAddress	Address in the server to read from.
	\param[in] 	Unit	Identity of the unit (0-255) in the server.
	\param[out] UpdateDone	When the function has completed succesfully, this value is set to TRUE.
	\param[out] Active	Set to TRUE when function is active.
	\param[out] Busy	Set to TRUE when function is accessing the server.
	\param[out] Error	If an error occurs while exeuting the function, this output is set to TRUE.
	\param[out] ErrorID	Error number from the function block.
	\param[out] Status	Normally set to zero otherwise something is wrong or function are waiting to get completed.
*/
void MB_PollDiscreteInputs(struct MB_PollDiscreteInputs* inst)
{
	CHECK_INPUT_QUANTITY_CYCLIC_MACRO(BRSE_MB_MAX_DISCRETE_INPUTS)
	EXEC_MODBUS_CYCLIC_FUNCTION_MACRO(BRSE_MB_READ_DISCRETE_INPUTS, inst->PollInterval)
}
```

#### Version_History.c
```c
/*!
\page History

\section History

\par V0.00
	\arg First draft version

\par V1.00
	\arg First functional version. Added inline comments.

\par V1.01
	\arg Added the input Unit in the client requests. Make it possible to communicate to many units in the same server in a simple way.
	\arg Added documentation for the client.

\par V1.02
	\arg Updated documentation.

\par V1.03
	\arg Added functionality for handling 4 byte variables.

\par V1.10
	\arg Release version for handling 4 byte holding registers

\par V1.11
	\arg Bugfix for writing multiple holding registers 4 byte. the last INT was copied in the wrong way.

\par V1.12
	\arg Bugfixes:
	\arg Allocation functions, if allocation failed, write to logbook and don't memset.
	\arg WriteHoldingRegister, 4WriteByteHoldingRegisters, WriteCoils buffer lengths were 1 byte too long.
	\arg Client functions check if the queue is alive while waiting for answers, returning error codes if the queue died.

\par V1.13
	\arg Minor change in the poll macro (client). Previously the condition to execute was (cycleCounter%pollCycles==0), now it's cycleCounter>=pollCycles (cycleCounter is reset when command is executed).

\par V1.14
	\arg Pagefault when writing to a single holding register when this was mapped as a 4-byte value has been fixed. Now
	an ILLEGAL_DATA_ADDRESS is returned if a 4byte value is mapped on that modbus reference.
	\arg All function blocks with an \b Execute input have been changed so that the execute input is edge sensitive (previously,
	the input was handled rather as an \b Enable input)
	\arg MB_QUEUE_SIZE has been set up to 50, it seems unlikely to have more simultaneous function calls than this at the moment.
	\arg Added dependency to the brsystem library, which reads out the cycle time of the task. The inputs of the functions have therefore changed from \b Poll/PushCycles to \b Poll/PushInterval, which you specify in ms.

\par V1.15
	\arg Corrected status bits from push and poll functions.

\par V1.16
	\arg MB_AllocClient : Changed return value to always return the internal address, even though allocation has already been performed.
	\arg Added extra information on the Error_Number page
	\arg Added the ModbusUDP adapter library BRSE_MBU to the documentation
*/
```

### Library Logical/ExtPack/_Comms/ModbusComms/ModbusComms_v1/Libraries/BRSE_MBT (ANSIC, version 1.21.1)
Depends on: BRSE_MB, astcp, sys_lib, AsString, brsystem, AsIecCon, standard

#### BRSE_MBT.typ - Exported data types
```iecst
TYPE
	BRSE_MBT_ReceiveBuff_typ : 	STRUCT
		Byte : ARRAY[0..BRSE_MBT_MAX_BUFFER]OF USINT;
	END_STRUCT;
	BRSE_MBT_ClientInfo_typ : 	STRUCT
		Ident : UDINT;
		Port : UINT;
		IpAddr : ARRAY[0..17]OF USINT;
	END_STRUCT;
	BRSE_MBT_ClientRequest_typ : 	STRUCT
		TransactionId : UINT;
		ProtocolId : UINT;
		Length : UINT;
	END_STRUCT;
	BRSE_MBT_Internal_typ : 	STRUCT
		TcpOpenIdent : UDINT;
	END_STRUCT;
	MBT_ClientInternal_typ : 	STRUCT
		TcpOpenIdent : ARRAY[0..MB_MAX_CLIENTS]OF UDINT;
	END_STRUCT;
	BRSE_MBT_Client_typ : 	STRUCT
		Info : BRSE_MBT_ClientInfo_typ;
		Request : BRSE_MBT_ClientRequest_typ;
		RecvBuffer : ARRAY[0..BRSE_MBT_MAX_BUFFER]OF USINT;
		SendBuffer : ARRAY[0..BRSE_MBT_MAX_BUFFER]OF USINT;
		FB_TcpRecv : TcpRecv;
		FB_TcpSend : TcpSend;
		FB_TcpIoctl : TcpIoctl;
		ResponseByteSize : UINT;
		State : USINT; (*0=no client, 1=receiving, 2=sending, 9=disconnecting*)
		TON_Disconnect : TON;
	END_STRUCT;
	BRSE_MBT_NewClient_typ : 	STRUCT
		IpAddr : ARRAY[0..17]OF USINT;
		CloseIdent : UDINT;
		ReconnectClientIdx : UINT;
		ReconnectClient : BOOL;
	END_STRUCT;
END_TYPE
```

#### BRSE_MBT_Server.c
```c
/*! \file BRSE_MBT_Server.c */

#include "BRSE_MBT.h"
#include "BRSE_MBT_Main.h"

#ifdef _SG4
	#define SWAPUINT	swapUINT
	#define SWAPINT		swapINT
#else
	#define SWAPUINT
	#define SWAPINT
#endif

#define	BUSY			65535
#define DISABLED		65534

/* B&R Modbus TCP Server */
/* (spec: http://www.rtaautomation.com/modbustcp/files/Open_ModbusTCP_Standard.pdf)
 *
 * Listens to port 502 for connecting clients. Responds to tcp requests according to specification.
 *
 * byte 0:  transaction identifier - copied by server - usually 0
 * byte 1:  transaction identifier - copied by server - usually 0
 * byte 2:  protocol identifier = 0
 * byte 3:  protocol identifier = 0
 * byte 4:  length field (upper byte) = 0 (since all messages are smaller than 256)
 * byte 5:  length field (lower byte) = number of bytes following
 * byte 6: 	unit identifier (previously 'slave address')
 *
 * byte 7: 	MODBUS function code
 * byte 8 	on:         data as needed
*/

BRSE_MBT_Internal_typ BRSE_MBT_ServerInternal;

UDINT MBT_GetServerInternalStructAddr()
{
	return (UDINT) &BRSE_MBT_ServerInternal;
}

/*!
	\interface BRSE_MBT_Server
	\brief Server: Create a connection to a physical Ethernet Port and open port 502 and starts	listen for incoming modbus messages.

	\param[in]	Enable	Enables execution of the function.
	\param[in]	ClientFormat	Set the format of 4 byte variables to Intel or Motorola. BRSE_MB_INTEL / BRSE_MB_MOTOROLA
	\param[in]	SocketTimeout	Time in seconds that the system keeps the socket alive after closing it (linger time). This can be used as the opposite station still has some data to send. If the input is zero the socket is closed immediately.
	\param[out] Status	Return status.

*/
void BRSE_MBT_Server(struct BRSE_MBT_Server* inst)
{
	UINT clientIdx;

	switch (inst->Step)
	{
		case  0 : /* init */
			inst->FB_TcpOpen.pIfAddr = 0;
			inst->FB_TcpOpen.port = inst->Port;
			inst->FB_TcpOpen.options = tcpOPT_REUSEADDR;
			inst->Error = 0;
			if (inst->Enable)
			{
				inst->Step = 10;
			}
			break;

		case 10: /* Open port */
			inst->FB_TcpOpen.enable = 1;
			TcpOpen(&inst->FB_TcpOpen);
			if (inst->FB_TcpOpen.status == 0)
			{
				inst->FB_TcpServer.enable = 1;
				inst->FB_TcpServer.ident = inst->FB_TcpOpen.ident;
				inst->FB_TcpServer.backlog = 0;
				inst->FB_TcpServer.pIpAddr = (UDINT)inst->NewClient.IpAddr;
				BRSE_MBT_ServerInternal.TcpOpenIdent = inst->FB_TcpOpen.ident;
				inst->Step = 15; /* wait for request */
			}
			else if (inst->FB_TcpOpen.status != BUSY)
			{
				/*inst->Step = 70;*/
			}
			break;

		case 15: /* Disabled */
			if (inst->Enable)
			{
				inst->Step = 20;
			}
			break;

		case 20: /* Read requests and respond */
			inst->IsBusy = 0;

			/* Check if any connections are to be closed */
			if (inst->NewClient.CloseIdent != 0) /* Close an old client connection (client has reconnected) */
			{
				inst->FB_TcpCloseOld.enable = 1;
				inst->FB_TcpCloseOld.ident	= inst->NewClient.CloseIdent;
				inst->FB_TcpCloseOld.how = 0; /*tcpSHUT_RD | tcpSHUT_WR;*/
				TcpClose(&inst->FB_TcpCloseOld);
				if(inst->FB_TcpCloseOld.status != BUSY) /* Nevermind errors here */
				{
					inst->NewClient.CloseIdent = 0;

					if(inst->FB_TcpCloseOld.status)
					{
						strcpy(inst->Log[inst->LogIndex], "Close1 error: ");
						itoa(inst->FB_TcpCloseOld.status, (UDINT)inst->TmpStr);
						strcat(inst->Log[inst->LogIndex], inst->TmpStr);
						strcat(inst->Log[inst->LogIndex], " id: ");
						itoa(inst->FB_TcpCloseOld.ident, (UDINT)inst->TmpStr);
						strcat(inst->Log[inst->LogIndex], inst->TmpStr);
						inst->LogIndex++;
					}

				}
				inst->IsBusy = inst->IsBusy || inst->FB_TcpCloseOld.status == BUSY;
			}
			else
			{
				for(clientIdx = 0; clientIdx<BRSE_MBT_MAX_CLIENT; clientIdx++) /* Loop through clients and see if they are to be closed */
				{
					if (inst->Clients[clientIdx].State == 99)
					{
						inst->FB_TcpClose[clientIdx].enable = 1;
						inst->FB_TcpClose[clientIdx].ident	= inst->Clients[clientIdx].Info.Ident;
						inst->FB_TcpClose[clientIdx].how = 0;/* tcpSHUT_RD | tcpSHUT_WR;*/
						TcpClose(&inst->FB_TcpClose[clientIdx]);
						if(inst->FB_TcpClose[clientIdx].status != BUSY) /* Nevermind errors here */
						{
							if(inst->FB_TcpClose[clientIdx].status)
							{
								strcpy(inst->Log[inst->LogIndex], "Close2 error: ");
								itoa(inst->FB_TcpClose[clientIdx].status, (UDINT)inst->TmpStr);
								strcat(inst->Log[inst->LogIndex], inst->TmpStr);
								strcat(inst->Log[inst->LogIndex], " id: ");
								itoa(inst->FB_TcpClose[clientIdx].ident, (UDINT)inst->TmpStr);
								strcat(inst->Log[inst->LogIndex], inst->TmpStr);
								inst->LogIndex++;
							}

							BRSE_MBT_RemoveClient(inst, clientIdx);

						}
						inst->IsBusy = inst->IsBusy || inst->FB_TcpClose[clientIdx].status == BUSY;
						break; /* break for-loop; can only run TcpClose on one client at a time */
					}
				}
			}

			/* Check for new clients if maximum nbr of clients has not been reached */
			if (inst->ClientNr < BRSE_MBT_MAX_CLIENT && (inst->Error==0 || inst->FB_TcpServer.status == BUSY))
			{
				TcpServer(&inst->FB_TcpServer);
				if (inst->FB_TcpServer.status == 0) /* client connected */
				{
					BRSE_MBT_AddClient(inst);
				}
				else if (inst->FB_TcpServer.status == tcpERR_INVALID_IDENT ||
						inst->FB_TcpServer.status == tcpERR_SOCKET_LISTEN)
				{
					inst->Error = inst->FB_TcpServer.status;
					if (inst->LogIndex < BRSE_MBT_LOG_MAX)
					{
						strcpy(inst->Log[inst->LogIndex], "Server error: ");
						itoa(inst->FB_TcpServer.status, (UDINT)inst->TmpStr);
						strcat(inst->Log[inst->LogIndex], inst->TmpStr);
						strcat(inst->Log[inst->LogIndex], " ");
						inst->LogIndex++;
					}
				}/* inst->FB_TcpServer.status == tcpERR_SOCKET_ACCEPT inst->FB_TcpServer.status == tcpERR_NOMORE_IDENTS ||*/
				inst->IsBusy = inst->IsBusy || (inst->FB_TcpServer.status == BUSY);
			}

			/* Loop through clients, respond to any requests */
			for(clientIdx = 0; clientIdx < BRSE_MBT_MAX_CLIENT; clientIdx++)
			{
				switch(inst->Clients[clientIdx].State)
				{
					case 0: /* No client initialized */
						break;

					case 1:
						inst->Clients[clientIdx].State = 10;
						break;

					case 10: /* Set linger options */
						inst->LingerOptions.lOnOff = 1;
						inst->LingerOptions.lLinger = inst->SocketTimeout;
						inst->Clients[clientIdx].FB_TcpIoctl.enable = 1;
						inst->Clients[clientIdx].FB_TcpIoctl.ident = inst->Clients[clientIdx].Info.Ident;
						inst->Clients[clientIdx].FB_TcpIoctl.pData = (UDINT)&inst->LingerOptions;
						inst->Clients[clientIdx].FB_TcpIoctl.datalen = sizeof(inst->LingerOptions);
						inst->Clients[clientIdx].FB_TcpIoctl.ioctl = tcpSO_LINGER_SET;
						TcpIoctl(&inst->Clients[clientIdx].FB_TcpIoctl);
						if (inst->Clients[clientIdx].FB_TcpIoctl.status != BUSY)
						{
							inst->Clients[clientIdx].State = 11;
						}
						break;

					case 11: /* catch errors */
						if (inst->Error == 0 && inst->Enable)
							inst->Clients[clientIdx].State = 2;
						else
							break;

					case 2: /* Receive */
						TcpRecv(&inst->Clients[clientIdx].FB_TcpRecv);
						if (inst->Clients[clientIdx].FB_TcpRecv.status == BUSY ||
						inst->Clients[clientIdx].FB_TcpRecv.status == DISABLED ||
						inst->Clients[clientIdx].FB_TcpRecv.status == tcpERR_NO_DATA)
						{
							; /* No data received */
						}
						else if (inst->Clients[clientIdx].FB_TcpRecv.status == tcpERR_NOT_CONNECTED ||
							inst->Clients[clientIdx].FB_TcpRecv.status != 0) /* If any error, typically if client disconnected, remove client */
						{
							inst->Clients[clientIdx].State = 99; /* Disconnect client */
						}
						else if (inst->Clients[clientIdx].FB_TcpRecv.status == 0) /* Frame received */
						{
							inst->Clients[clientIdx].ResponseByteSize = BRSE_MBT_AnalyzeReqFromClient(inst, clientIdx);
							if (inst->Clients[clientIdx].ResponseByteSize > 0)
							{
								inst->Clients[clientIdx].FB_TcpSend.datalen = inst->Clients[clientIdx].ResponseByteSize;
								inst->Clients[clientIdx].State = 3; /* Send response */
							}
							else /* Client has disconnected */
 							{
								inst->Clients[clientIdx].State = 99;
							}
							/* Fall through! */
						}
						inst->IsBusy = inst->IsBusy || inst->Clients[clientIdx].FB_TcpRecv.status == BUSY;
						if (inst->Clients[clientIdx].State != 3)
							break;
						/* Beware! Fall through if state is 3 */

					case 3: /* Send response */
						TcpSend(&inst->Clients[clientIdx].FB_TcpSend);
						if( (inst->Clients[clientIdx].FB_TcpSend.status == BUSY	) 	||
							(inst->Clients[clientIdx].FB_TcpSend.status == DISABLED)||
							(inst->Clients[clientIdx].FB_TcpSend.status == tcpERR_SENTLEN)	)
						{
							;
						}
						else if(inst->Clients[clientIdx].FB_TcpSend.status != 0) /* Disconnect client */
						{
							if (inst->LogIndex < BRSE_MBT_LOG_MAX)
							{
								strcpy(inst->Log[inst->LogIndex], "TcpSend error: ");
								itoa(inst->Clients[clientIdx].FB_TcpSend.status, (UDINT)inst->TmpStr);
								strcat(inst->Log[inst->LogIndex], inst->TmpStr);
								strcat(inst->Log[inst->LogIndex], " ");
								strcat(inst->Log[inst->LogIndex], inst->Clients[clientIdx].Info.IpAddr);
								inst->LogIndex++;
							}
							inst->Clients[clientIdx].State = 99;
						}
						else /* Back to receive */
						{
							memset(inst->Clients[clientIdx].RecvBuffer, 0, sizeof(inst->Clients[clientIdx].RecvBuffer));
							memset(inst->Clients[clientIdx].SendBuffer, 0, sizeof(inst->Clients[clientIdx].SendBuffer));
							inst->Clients[clientIdx].State = 2;
						}
						inst->IsBusy = inst->IsBusy || inst->Clients[clientIdx].FB_TcpSend.status == BUSY;
						break;
				}
			}

			if (!inst->IsBusy && inst->Error != 0)
			{
				inst->Step = 70;
			}
			else if (!inst->Enable && !inst->IsBusy) /* If disabled, move to idle */
			{
				if (inst->LogIndex < BRSE_MBT_LOG_MAX && inst->Step != 15)
				{
					strcpy(inst->Log[inst->LogIndex], "FUB Disabled. Go to idle");
					inst->LogIndex++;
				}
				inst->Step = 15; /* idle */
			}
			break;

		case 70:	/* Error: close server connection */
			inst->FB_TcpCloseServer.enable = 1;
			inst->FB_TcpCloseServer.ident	= BRSE_MBT_ServerInternal.TcpOpenIdent;
			inst->FB_TcpCloseServer.how = 0; /*tcpSHUT_RD | tcpSHUT_WR;*/
			TcpClose(&inst->FB_TcpCloseServer);
			if(inst->FB_TcpCloseServer.status != BUSY)
			{
				/* Remove all clients */
				for (clientIdx = 0 ; clientIdx<BRSE_MBT_MAX_CLIENT ; clientIdx++)
				{
					BRSE_MBT_RemoveClient(inst, clientIdx);
				}
				inst->ClientNr = 0;
				inst->Step = 0;
				BRSE_MBT_ServerInternal.TcpOpenIdent = 0;
				if (inst->LogIndex < BRSE_MBT_LOG_MAX)
				{
					strcpy(inst->Log[inst->LogIndex], "Disconnect server: ");
					itoa(inst->FB_TcpCloseServer.status, (UDINT)inst->TmpStr);
					strcat(inst->Log[inst->LogIndex], inst->TmpStr);
					strcat(inst->Log[inst->LogIndex], " ");
					inst->LogIndex++;
				}
			}
			break;

	}
	if (inst->LogIndex == BRSE_MBT_LOG_MAX)
	{
		inst->LogIndex = 0;
	}
	strcpy(inst->Log[inst->LogIndex], "");

	//Disconnect old inactive clients
	for(clientIdx = 0; clientIdx<BRSE_MBT_MAX_CLIENT; clientIdx++) /* Loop through clients and see if they are to be closed */
	{
		inst->Clients[clientIdx].TON_Disconnect.PT = BRSE_DISCONNECT_TIMEOUT;
		if (inst->Clients[clientIdx].State == 2 )
		{
			inst->Clients[clientIdx].TON_Disconnect.IN = 1;
		}
		else
		{
			 inst->Clients[clientIdx].TON_Disconnect.IN = 0;
		}
		if (inst->Clients[clientIdx].TON_Disconnect.Q)	//Close client
		{
			inst->Clients[clientIdx].TON_Disconnect.IN = 0;
			inst->Clients[clientIdx].State = 99;
		}
		TON(&inst->Clients[clientIdx].TON_Disconnect);
	}
}

/* Returns number of bytes in possible response message */
UINT BRSE_MBT_AnalyzeReqFromClient(struct BRSE_MBT_Server* inst, UINT clientIdx)
{
	UINT uintVar;
	UINT length;

	/* Check for tcp length errors */
	if (inst->Clients[clientIdx].FB_TcpRecv.recvlen == 0) /* client closed the connection */
	{
		return 0;
	}
	else if (inst->Clients[clientIdx].FB_TcpRecv.recvlen < 8)
	{
		return BRSE_MBT_CreateErrorMessage(inst, BRSE_MB_ERR_ILLEGAL_DATA_VALUE, clientIdx);
	}
	else if (inst->Clients[clientIdx].FB_TcpRecv.recvlen > BRSE_MBT_MAX_BUFFER)
	{
		return BRSE_MBT_CreateErrorMessage(inst, BRSE_MB_ERR_ILLEGAL_RESPONSE_LEN, clientIdx);
	}

	/* Parse tcp message information. Byte 0-5 */
	memcpy(&uintVar, &(inst->Clients[clientIdx].RecvBuffer[0]), sizeof(uintVar));
	inst->Clients[clientIdx].Request.TransactionId = SWAPUINT(uintVar);
	memcpy(&uintVar, &(inst->Clients[clientIdx].RecvBuffer[2]), sizeof(uintVar));
	inst->Clients[clientIdx].Request.ProtocolId = SWAPUINT(uintVar);
	memcpy(&uintVar,&(inst->Clients[clientIdx].RecvBuffer[4]), sizeof(uintVar));
	inst->Clients[clientIdx].Request.Length = SWAPUINT(uintVar);

	/* Validate tcp message information */
	if(	(inst->Clients[clientIdx].Request.ProtocolId	!= 0) || (inst->Clients[clientIdx].Request.Length == 0))
	{
		return BRSE_MBT_CreateErrorMessage(inst, BRSE_MB_ERR_ILLEGAL_DATA_VALUE, clientIdx);
	}

	/* Run message through MB_Server. Byte 6 is unit id. */
	inst->FB_BRSE_MB_Server.Unit = inst->Clients[clientIdx].RecvBuffer[6];
	inst->FB_BRSE_MB_Server.ClientFormat = inst->ClientFormat;
	memcpy(inst->FB_BRSE_MB_Server.InputBuffer, &(inst->Clients[clientIdx].RecvBuffer[7]), 254); /* 254 is sizeof input buffer */
	BRSE_MB_Server(&inst->FB_BRSE_MB_Server);

	/* Check for message errors */
	if (inst->FB_BRSE_MB_Server.Status == BRSE_MB_ERR_ILLEGAL_FUNCTION)
		return BRSE_MBT_CreateErrorMessage(inst, BRSE_MB_ERR_ILLEGAL_FUNCTION, clientIdx);
	else if (inst->FB_BRSE_MB_Server.Status == BRSE_MB_ERR_ILLEGAL_DATA_ADDRESS)
		return BRSE_MBT_CreateErrorMessage(inst, BRSE_MB_ERR_ILLEGAL_DATA_ADDRESS, clientIdx);
	else if (inst->FB_BRSE_MB_Server.Status == BRSE_MB_ERR_ILLEGAL_DATA_VALUE)
		return BRSE_MBT_CreateErrorMessage(inst, BRSE_MB_ERR_ILLEGAL_DATA_VALUE, clientIdx);
	else if (inst->FB_BRSE_MB_Server.Status == BRSE_MB_ERR_ILLEGAL_RESPONSE_LEN)
		return BRSE_MBT_CreateErrorMessage(inst, BRSE_MB_ERR_ILLEGAL_RESPONSE_LEN, clientIdx);
	else if (inst->FB_BRSE_MB_Server.Status != 0)
		return BRSE_MBT_CreateErrorMessage(inst, BRSE_MB_ERR_ILLEGAL_DATA_VALUE, clientIdx);

	/* Message ok. Create response */
	/* Transaction id: 2 byte */
	memcpy(&inst->Clients[clientIdx].SendBuffer[0], &inst->Clients[clientIdx].RecvBuffer[0], sizeof(uintVar));
	/* Protocol id: 2 byte */
	memcpy(&inst->Clients[clientIdx].SendBuffer[2], &inst->Clients[clientIdx].RecvBuffer[2], sizeof(uintVar));
	/* Length: 2 byte */
	length = 1 + inst->FB_BRSE_MB_Server.BufferLength; /* The extra byte is the unit identifier */
	uintVar = SWAPUINT(length);
	memcpy(&inst->Clients[clientIdx].SendBuffer[4], &uintVar, sizeof(uintVar));
	/* Unit: 1 byte */
	inst->Clients[clientIdx].SendBuffer[6] = inst->Clients[clientIdx].RecvBuffer[6];
	/* Message response */
	memcpy(&inst->Clients[clientIdx].SendBuffer[7], &inst->FB_BRSE_MB_Server.OutputBuffer[0], 254);
	return 7 + inst->FB_BRSE_MB_Server.BufferLength; /* Number of bytes to be sent */
}

UINT BRSE_MBT_AddClient(struct BRSE_MBT_Server* inst)
{
	INT index = -1;
	UINT i = 0;

	if (inst->ClientNr < BRSE_MBT_MAX_CLIENT)
	{
		/* Check if client has already connedted before */
		for (i=0; i < BRSE_MBT_MAX_CLIENT; i++)
		{
			/* Check if client was already connected, in that case: reconnect that client */
			if (inst->Clients[i].Info.Ident != 0 && !memcmp(inst->Clients[i].Info.IpAddr, inst->NewClient.IpAddr, sizeof(inst->NewClient.IpAddr)) && inst->FB_TcpServer.identclnt == inst->Clients[i].Info.Ident )
			{
				inst->NewClient.CloseIdent = inst->Clients[i].Info.Ident; /* Make sure the old client handle gets closed */
				BRSE_MBT_RemoveClient(inst, i);
				index = i;
			}
		}
		/* New client */
		if (index < 0)
		{
			/* Find first avilable index */
			for (i=0; i < BRSE_MBT_MAX_CLIENT; i++)
			{
				if (index<0 && inst->Clients[i].Info.Ident == 0)
				{
					index=i;
				}
			}
		}
		if (index<0) /* No more clients allowed */
			return BRSE_MBT_ERR_TOO_MANY_CLIENTS;

		/* Save client info */
		inst->Clients[index].Info.Ident = inst->FB_TcpServer.identclnt;
		inst->Clients[index].Info.Port = inst->FB_TcpServer.portclnt;
		memcpy(inst->Clients[index].Info.IpAddr, inst->NewClient.IpAddr, sizeof(inst->NewClient.IpAddr));

		/* Initialize TcpRecv */
		inst->Clients[index].FB_TcpRecv.enable = 1;
		inst->Clients[index].FB_TcpRecv.ident = (UDINT)inst->FB_TcpServer.identclnt;
		inst->Clients[index].FB_TcpRecv.pData = (UDINT)inst->Clients[index].RecvBuffer;
		inst->Clients[index].FB_TcpRecv.datamax = BRSE_MBT_MAX_BUFFER+1;
		inst->Clients[index].FB_TcpRecv.flags = 0;

		/* Initialize TcpSend */
		inst->Clients[index].FB_TcpSend.enable = 1;
		inst->Clients[index].FB_TcpSend.flags = 0;
		inst->Clients[index].FB_TcpSend.ident = (UDINT)inst->FB_TcpServer.identclnt;
		inst->Clients[index].FB_TcpSend.pData = (UDINT)inst->Clients[index].SendBuffer;

		/* Client counter */
		inst->ClientNr++;

		/* Start receiving data */
		inst->Clients[index].State = 1;

		/* Write log message */
		if (inst->LogIndex < BRSE_MBT_LOG_MAX)
		{
			memset(inst->Log[inst->LogIndex], 0, sizeof(inst->Log[inst->LogIndex]));
			memcpy(inst->Log[inst->LogIndex], inst->NewClient.IpAddr, sizeof(inst->NewClient.IpAddr));
			strcat(inst->Log[inst->LogIndex], " connected on id:");
			itoa(inst->FB_TcpServer.identclnt, (UDINT)inst->TmpStr);
			strcat(inst->Log[inst->LogIndex], inst->TmpStr);
			inst->LogIndex++;
		}
		return 0;
	}
	else
	{
		return BRSE_MBT_ERR_TOO_MANY_CLIENTS;
	}
	return 0;
}

void BRSE_MBT_RemoveClient(struct BRSE_MBT_Server* inst, UINT clientIdx)
{
	if (inst->ClientNr > 0)
	{
		if (inst->LogIndex < BRSE_MBT_LOG_MAX)
		{
			memset(inst->Log[inst->LogIndex], 0, sizeof(inst->Log[inst->LogIndex]));
			memcpy(inst->Log[inst->LogIndex], inst->Clients[clientIdx].Info.IpAddr, sizeof(inst->Clients[clientIdx].Info.IpAddr));
			strcat(inst->Log[inst->LogIndex], " removed");
			inst->LogIndex++;
		}
		inst->Clients[clientIdx].FB_TcpRecv.enable = 0;
		inst->Clients[clientIdx].FB_TcpSend.enable = 0;
		inst->Clients[clientIdx].State = 0;
		inst->Clients[clientIdx].Info.Ident = 0;
		memset(inst->Clients[clientIdx].Info.IpAddr, 0, sizeof(inst->Clients[clientIdx].Info.IpAddr));
		inst->Clients[clientIdx].Info.Port = 0;
		memset(inst->Clients[clientIdx].SendBuffer, 0, sizeof(inst->Clients[clientIdx].SendBuffer));
		memset(inst->Clients[clientIdx].RecvBuffer, 0, sizeof(inst->Clients[clientIdx].RecvBuffer));
		inst->ClientNr--;
	}
}

UINT BRSE_MBT_CreateErrorMessage(struct BRSE_MBT_Server* inst, UINT errorCode, UINT clientIdx)
{
	UINT	length;
	UINT	uintVar;

	memset(inst->Clients[clientIdx].SendBuffer, 0, sizeof(inst->Clients[clientIdx].SendBuffer));
	/* Transaction id: 2 byte */
	uintVar = SWAPUINT(inst->Clients[clientIdx].Request.TransactionId);
	memcpy(&inst->Clients[clientIdx].SendBuffer[0], &inst->Clients[clientIdx].RecvBuffer[0], sizeof(uintVar));
	/* Protocol id: 2 byte */
	uintVar = SWAPUINT(inst->Clients[clientIdx].Request.ProtocolId);
	memcpy(&inst->Clients[clientIdx].SendBuffer[2], &inst->Clients[clientIdx].RecvBuffer[2], sizeof(uintVar));
	/* Length: 2 byte */
	length = 3;
	uintVar = SWAPUINT(length);
	memcpy(&inst->Clients[clientIdx].SendBuffer[4], &uintVar, sizeof(uintVar));
	/* Unit: 1 byte */
	inst->Clients[clientIdx].SendBuffer[6] = inst->Clients[clientIdx].RecvBuffer[6];
	/* Function code: 1 byte */
	inst->Clients[clientIdx].SendBuffer[7] = inst->Clients[clientIdx].RecvBuffer[7] +  0x80;
	/* Exception code: 1 byte */
	inst->Clients[clientIdx].SendBuffer[8] = errorCode;
	return 9;
}

/*!
	\interface MBT_ServerExit
	\brief Server: Closes open tcp ports. Use this in the exit routine of the program.

	\param[out] Status	Return status.

*/
void MBT_ServerExit(struct MBT_ServerExit* inst)
{
	if (BRSE_MBT_ServerInternal.TcpOpenIdent != 0)
	{
		inst->FB_TcpClose.enable = 1;
		inst->FB_TcpClose.ident	= BRSE_MBT_ServerInternal.TcpOpenIdent;
		inst->FB_TcpClose.how = tcpSHUT_RD | tcpSHUT_WR;
		TcpClose(&inst->FB_TcpClose);
		if(inst->FB_TcpClose.status != BUSY)
		{
			BRSE_MBT_ServerInternal.TcpOpenIdent = 0;
		}
	}
}
```

#### Example_Client.c
```c
/*!

 \page Example_client Example Client
 \section Example_client Example Client

 \par Description
	This program set up an TCP modbus client on the ethernet port of the system.
	The client can use both event driven and cyclic operation, in this example both are used.
	To send and recive the event driven variables startMotor and motorRunning the variable sendToServer need to be forced to TRUE.
	The variables setSpeed and actSpeed are automaticly updated every 200 taskcycle.

 \par Example
  Example \ref tasks can be found here.

\par MBclient.var
\code
VAR
	FB_MB_WriteCoils : MB_WriteCoils := (0);
	FB_MB_ReadDiscreteInputs : MB_ReadDiscreteInputs := (0);
	FB_MB_PushHoldingRegisters : MB_PushHoldingRegisters := (0);
	FB_MB_PollInputRegisters : MB_PollInputRegisters := (0);
	FB_MB_Poll4ByteHoldingRegisters : MB_Poll4ByteHoldingRegisters := (0);
	FB_MBT_Client : MBT_Client := (0);
	FB_MBT_ExitClient : MBT_ExitClient := (0);
	startMotor : ARRAY[0..2] OF BOOL := [3(FALSE)];
	motorRunning : ARRAY[0..2] OF BOOL := [3(FALSE)];
	setSpeed : ARRAY[0..2] OF INT := [3(0)];
	actSpeed : ARRAY[0..2] OF INT := [3(0)];
	actTemp : ARRAY[0..3] OF REAL := [4(0.0)];
	sendToServer : BOOL := FALSE;
	state : USINT := 0;
END_VAR
\endcode

\par MBclient.st
\code
PROGRAM _INIT

	MB_AllocClient(1);								(* Create a Modbus client with identity = 1 *)

	FB_MB_WriteCoils.ClientID			:= 1;				(* Identity created in AllocClient *)
	FB_MB_WriteCoils.Execute			:= 0;				(* Do not execute function block yet *)
	FB_MB_WriteCoils.Quantity			:= 3;				(* Number of register to write *)
	FB_MB_WriteCoils.VariablesAddress		:= ADR(startMotor[0]);		(* Address of the BOOL variable *)
	FB_MB_WriteCoils.StartAddress			:= 0;				(* Address in the server to write to *)
	FB_MB_WriteCoils.Unit				:= 0;				(* Unit identity in the server *)

	FB_MB_ReadDiscreteInputs.ClientID		:= 1;				(* Identity created in AllocClient *)
	FB_MB_ReadDiscreteInputs.Execute		:= 0;				(* Do not execute function block yet *)
	FB_MB_ReadDiscreteInputs.Quantity		:= 3;				(* Number of register to read *)
	FB_MB_ReadDiscreteInputs.VariablesAddress	:= ADR(motorRunning[0]);	(* Address of the BOOL variable *)
	FB_MB_ReadDiscreteInputs.StartAddress		:= 0;				(* Address in the server to read from *)
	FB_MB_ReadDiscreteInputs.Unit			:= 0;				(* Unit identity in the server *)

	FB_MB_PushHoldingRegisters.ClientID		:= 1;				(* Identity created in AllocClient *)
	FB_MB_PushHoldingRegisters.Enable		:= 0;				(* Do not enable function block yet *)
	FB_MB_PushHoldingRegisters.Quantity		:= 3;				(* Number of register to write *)
	FB_MB_PushHoldingRegisters.PushCycles		:= 200;				(* Number of cycles between write requests *)
	FB_MB_PushHoldingRegisters.VariablesAddress	:= ADR(setSpeed[0]);		(* Address of the INT variable *)
	FB_MB_PushHoldingRegisters.StartAddress		:= 0;				(* Address in the server to write to *)
	FB_MB_PushHoldingRegisters.Unit			:= 0;				(* Unit identity in the server *)

	FB_MB_PollInputRegisters.ClientID		:= 1;				(* Identity created in AllocClient *)
	FB_MB_PollInputRegisters.Enable			:= 0;				(* Do not enable function block yet *)
	FB_MB_PollInputRegisters.Quantity		:= 3;				(* Number of register to read *)
	FB_MB_PollInputRegisters.PushCycles		:= 200;				(* Number of cycles between read requests *)
	FB_MB_PollInputRegisters.VariablesAddress	:= ADR(actSpeed[0]);		(* Address of the INT variable *)
	FB_MB_PollInputRegisters.StartAddress		:= 0;				(* Address in the server to read from *)
	FB_MB_PollInputRegisters.Unit			:= 0;				(* Unit identity in the server *)

	FB_MB_Poll4ByteHoldingRegisters.ClientID		:= 1;				(* Identity created in AllocClient *)
	FB_MB_Poll4ByteHoldingRegisters.Enable			:= 0;				(* Do not enable function block yet *)
	FB_MB_Poll4ByteHoldingRegisters.Quantity		:= 4;				(* Number of REAL values to read *)
	FB_MB_Poll4ByteHoldingRegisters.PushCycles		:= 200;				(* Number of cycles between read requests *)
	FB_MB_Poll4ByteHoldingRegisters.VariablesAddress:= ADR(actTemp[0]);	(* Address of the REAL variable *)
	FB_MB_Poll4ByteHoldingRegisters.StartAddress	:= 10;				(* Address in the server to read from *)
	FB_MB_Poll4ByteHoldingRegisters.Unit			:= 0;				(* Unit identity in the server *)

	FB_MBT_Client.ClientID				:= 1;				(* Identity created in AllocClient *)
	FB_MBT_Client.IpAddr				:= '10.46.10.153';		(* Ip address to the modbus server *)
	FB_MBT_Client.Port				:= 502;				(* Port on the modbus server *)
	FB_MBT_Client.CycleTime				:= 10;				(* The cycletime of the task in ms *)
	FB_MBT_Client.ServerFormat		:= BRSE_MB_INTEL; (* real values from server are in INTEL format *)

END_PROGRAM

PROGRAM _CYCLIC

	CASE state OF
		0 : (* Init step *)
			IF sendToServer = TRUE THEN
   				state := 10;
			END_IF

		10: (* Send coils to server and wait for response *)
			FB_MB_WriteCoils.Execute := TRUE;
			IF FB_MB_WriteCoils.Done OR FB_MB_WriteCoils.Error THEN
				FB_MB_WriteCoils.Execute := FALSE;
   				state := 20;
			END_IF

		20: (* Read the discreate inputs from server and wait for response *)
			FB_MB_ReadDiscreteInputs.Execute := TRUE;
   			IF FB_MB_ReadDiscreteInputs.Done OR FB_MB_ReadDiscreteInputs.Error THEN
				FB_MB_ReadDiscreteInputs.Execute := FALSE;
				state := 30;
			END_IF

		30: (* Start over again *)
			sendToServer := FALSE;
			state := 0;

	END_CASE;

	FB_MB_PollInputRegisters.Enable		:= 1;	(* Enable function block *)
	FB_MB_PushHoldingRegisters.Enable	:= 1;	(* Enable function block *)
	FB_MBT_Client.Enable			:= 1;	(* Enable function block *)

	FB_MB_WriteCoils();				(* Call function block *)
	FB_MB_ReadDiscreteInputs();			(* Call function block *)
	FB_MB_PollInputRegisters();			(* Call function block *)
	FB_MB_PushHoldingRegisters();			(* Call function block *)
	FB_MB_Poll4ByteHoldingRegisters();	(* Call function block *)

	FB_MBT_Client();				(* Call function block *)

END_PROGRAM

PROGRAM _EXIT

	(* Close the open tcp port *)
	FB_MBT_ExitClient(ClientID := 1);

END_PROGRAM

\endcode
*/

/*

Example on how to use the BRSE_MBT Library as a modbus client in C

#include <bur/plctypes.h>

#ifdef _DEFAULT_INCLUDES
 #include <AsDefault.h>
#endif

void _INIT MBRTestINIT( void )
{
	MB_AllocClient(4); // 4 is the client id

	MBT_Client_0.Enable = 1;
	MBT_Client_0.ClientID = 4;
	strcpy(MBT_Client_0.IpAddr, "192.168.0.1");
	MBT_Client_0.Port = 502;
	MBT_Client_0.Unit = 1;
	MBT_Client_0.CycleTime = 50;

	// Prepare to call any of the modbus master functions from the BRSE_MB library
	FB_MB_PushHoldingRegisters.ClientID = 2;
	FB_MB_PushHoldingRegisters.Enable = 1;
	FB_MB_PushHoldingRegisters.PushCycles = 300;
	FB_MB_PushHoldingRegisters.Quantity = 4;
	FB_MB_PushHoldingRegisters.StartAddress = 3;
	FB_MB_PushHoldingRegisters.VariablesAddress = (UDINT)&(IntArr[0]);
}

void _CYCLIC MBRTestCYCLIC( void )
{
	MB_PushHoldingRegisters(&MB_PushHoldingRegisters_0);
	MBT_Client(&MBT_Client_0);
}

*/
```

### Slave_mbus.var
```iecst
(********************************************************************
 * COPYRIGHT -- Bernecker + Rainer
 ********************************************************************
 * Program: Slave_mbus
 * File: Slave_mbus.var
 * Author: gimeneza
 * Created: March 07, 2017
 ********************************************************************
 * Local variables of program Slave_mbus
 ********************************************************************)
VAR
	FB_MBT_ServerExit : MBT_ServerExit := (0);
	i : UINT := 0;
	ident : USINT := 0;
END_VAR
```

### Program Logical/ExtPack/_Comms/SNTPClient/SNTPClient_v1/NwSNTPClient

#### TimeStateMachine.st
```iecst
ACTION TimeStateMachine:

	//Getting the TimeZoneId
	TimeZoneId;
	IF Network.Data.TimeZoneID<>TimeZoneId_copy THEN
		xNeedToResedTimeZoneId := TRUE;
		TimeZoneId_copy := Network.Data.TimeZoneID;
	END_IF

	CASE Time.State OF

		TIME_NOT_INITIALIZED:
			IF EDGEPOS(gPLC.xBlk_5s) THEN
				Network.Command.bCfgSetTimeZone := TRUE;
				Time.State := TIME_SETTING_TIMEZONE;
			END_IF

		TIME_SETTING_TIMEZONE:
			IF Network.Data.Step = 0 THEN
				Network.Command.bCfgSetSntpClient := TRUE;
				xNeedToResedTimeZoneId := FALSE;
				Time.Status.TimeUpdated := FALSE;
				Time.State := TIME_SETTING_CLIENT;
			END_IF

		TIME_SETTING_CLIENT:
			IF Network.Data.Step = 0 THEN
				IF Time.Params.DayLightSavingsTime THEN
					Network.Command.bGetTimeData := TRUE;
					Time.State := TIME_GETTING_TIMEDATA;
				ELSE
					Network.Command.bCfgGetSntpcData := TRUE;
					Time.State := TIME_RECEIVING_DATA;
				END_IF
			END_IF

		TIME_GETTING_TIMEDATA:
			IF Network.Data.Step = 0 THEN
				Network.Command.bCfgGetSntpcData := TRUE;
				Time.State := TIME_RECEIVING_DATA;
			END_IF

		TIME_RECEIVING_DATA:
			IF Network.Data.Step = 0 THEN
				Time.Status.TimeUpdated := TRUE;
				Time.State := TIME_IDLE;
			END_IF

		TIME_IDLE:
			//Modifyint ZoneId after changing the TimeZone
			IF xNeedToResedTimeZoneId THEN
				Network.Command.bCfgSetTimeZone := TRUE;
				Time.State := TIME_SETTING_TIMEZONE;
			END_IF

	END_CASE;

	//Defining value to Sw
	CASE Time.State OF
		TIME_NOT_INITIALIZED: Time.Status.SwState := 0;
		TIME_SETTING_TIMEZONE: Time.Status.SwState := 1;
		TIME_SETTING_CLIENT: Time.Status.SwState := 2;
		TIME_GETTING_TIMEDATA: Time.Status.SwState := 3;
		TIME_RECEIVING_DATA: Time.Status.SwState := 4;
		TIME_IDLE: Time.Status.SwState := 5;
	END_CASE;

END_ACTION
```

### Program Logical/ExtPack/_Cure/ArcLampGEW/ArcLampGew_v1/ArcLampGewCtrl (IEC)

#### Alarms.st
```iecst
ACTION Alarms:

	xAnyLampInError := FALSE;
	FOR iLamp:=1 TO data.Parameters.iLampQuantity DO
		IF data.Status.Lamps[iLamp].InAlarm AND data.Parameters.Lamps[iLamp].Enable THEN
			xAnyLampInError := TRUE;
		END_IF
	END_FOR;
	data.Status.xAnyLampInError := xAnyLampInError;

	IF Client.httpStatus = HTTPSTATUS_UNAUTORIZED THEN
		data.Alarms.Comms.xCredentialsError := TRUE;
	END_IF

	IF Client.httpStatus = HTTPSTATUS_INTERNALSERVERERROR THEN
		data.Alarms.Comms.xServerError := TRUE;
	END_IF

	IF data.Signals.In.xJam THEN
		data.Alarms.xJam := TRUE;
	END_IF

	/////////////////////////////////////////////////////////////////
	//  SOUND  SOUND  SOUND  SOUND  SOUND  SOUND  SOUND
	/////////////////////////////////////////////////////////////////

	arCommsError(xAlarm:= data.Alarms.xCommsError, xSilence:=data.Commands.xMute);
	arLampInError1(xAlarm:= data.Status.Lamps[1].InAlarm, xSilence:=data.Commands.xMute);
	arLampInError2(xAlarm:= data.Status.Lamps[2].InAlarm, xSilence:=data.Commands.xMute);
	arJam(xAlarm:= data.Alarms.xJam, xSilence:=data.Commands.xMute);

	reasonSound.0 := arCommsError.xAlarmSound;
	reasonSound.1 := arLampInError1.xAlarmSound;
	reasonSound.2 := arLampInError2.xAlarmSound;
	reasonSound.7 := arJam.xAlarmSound;

	data.AlSummary.xAlarmSound := reasonSound>0;

END_ACTION
```
